(* No error *)
	IF bError=FALSE THEN
		(*Event : Alarm*)
		IF strEventType='ALARM' THEN
			(*Set Alarm*)
			IF bEventSet=TRUE THEN
				GV_Events.aEventGroup[iEventGroup].aAlarm[iIdEvent].fbAlarm.Raise(0);
			ELSE
				GV_Events.aEventGroup[iEventGroup].aAlarm[iIdEvent].fbAlarm.Confirm(0);
				GV_Events.aEventGroup[iEventGroup].aAlarm[iIdEvent].fbAlarm.Clear(0,FALSE);
			END_IF
		END_IF
		(*Event : Message*)
		IF strEventType='MESSAGE' THEN
			GV_Events.aEventGroup[iEventGroup].aMessage[iIdEvent].fbMessage.Send(0);
		END_IF
		(*Event : OpMessage*)
		IF strEventType='OpMESSAGE' THEN
			(*Set Alarm*)
			IF bEventSet=TRUE THEN
				GV_Events.aEventGroup[iEventGroup].aOpMessage[iIdEvent].fbAlarm.Raise(0);
			ELSE
				GV_Events.aEventGroup[iEventGroup].aOpMessage[iIdEvent].fbAlarm.Confirm(0);
				GV_Events.aEventGroup[iEventGroup].aOpMessage[iIdEvent].fbAlarm.Clear(0,FALSE);
			END_IF
		END_IF
	END_IF

METHOD M_Event_Group_State
VAR_INPUT
	(** INT **)
	iEventGroup : INT ;
END_VAR
VAR_OUTPUT
	(** FLAG **)
	bEventPresence : BOOL ;
END_VAR
VAR
	(** INT **)
	iLoop : INT ;
END_VAR
//-----------------------------------------------------------------------------------------
//
//                  			M_Event_Group_State
//
//							Etat du groupe d'évènements  			
//-----------------------------------------------------------------------------------------
//
//Auteur: G.GOETZ (inspired by S.MANTZER)
//Création: 23.01.2026
//Dernière modification : 23.01.2026 (G.GOETZ)
//       			
//-----------------------------------------------------------------------------------------
//
//     							Liste des modifications  	
//
// 23.01.2026 (G.GOETZ) -> Création		
//-----------------------------------------------------------------------------------------

(* Initialized variables *)
bEventPresence:=FALSE;

(*Check if alarm activated in Group xx*)
FOR iLoop:=1 TO GV_Events.iMaxAlarms BY 1 DO
	IF GV_Events.aEventGroup[iEventGroup].aAlarm[iLoop].fbAlarm.eConfirmationState=2 THEN
		bEventPresence:=TRUE;
	END_IF;
END_FOR;
END_METHOD

END_FUNCTION_BLOCK

// ---- 02_Events/03_POUs/02_FBs/FB_Init_Call_Events.TcPOU
FUNCTION_BLOCK FB_Init_Call_Events
VAR_INPUT
END_VAR
VAR_OUTPUT
END_VAR
VAR
	(** FB **)
	fbInitEvents : FB_Init_Events ;
	fbEventGroupAssignement : FB_Event_Group_Number_Assignement ;
END_VAR

//-----------------------------------------------------------------------------------------
//
//                  			FB_Init_Call_Events
//
//					Gestion initialisation appel des évènements  			
//-----------------------------------------------------------------------------------------
//
//Auteur: G.GOETZ (inspired by S.MANTZER)
//Création: 21.01.2026
//Dernière modification : 21.01.2026 (G.GOETZ)
//       			
//-----------------------------------------------------------------------------------------
//
//     							Liste des modifications  	
//
// 21.01.2026 (G.GOETZ) -> Création		
//-----------------------------------------------------------------------------------------

// Alarms and Messages init
// Call first Event because we need to call one Event in the GUID to have it into .xml file
// Event group number assignment
fbEventGroupAssignement(iEventGroup:=GV_Events.iEventGroupCallEvent);
GV_Events.aEventGroup[GV_Events.iEventGroupCallEvent].aAlarm[1].fbAlarm.CreateEx(TC_Events.EventsAlarms.Alarm1,TRUE,0);
GV_Events.aEventGroup[GV_Events.iEventGroupCallEvent].aMessage[1].fbMessage.CreateEx(TC_Events.EventsMessages.Message1,0);

fbInitEvents(iEventGroup:=GV_Events.iEventGroupCallEvent, strEventType:='ALARM', strEventGuid:='784AC907-376D-4A8E-8897-3F447F113731', tcEventSeverity:=2);
fbInitEvents(iEventGroup:=GV_Events.iEventGroupCallEvent, strEventType:='MESSAGE', strEventGuid:='8930F18E-C6C1-418F-90B9-F30993F2C9E2', tcEventSeverity:=0);

END_FUNCTION_BLOCK

// ---- 02_Events/03_POUs/02_FBs/FB_Init_Events.TcPOU
FUNCTION_BLOCK FB_Init_Events
VAR_INPUT
	(** STRING **)	
	strEventType : STRING[20] ; // Type of the Event (ALARM or MESSAGE)
	strEventGuid : STRING[36] ; // Guid of the Event
	
	(** INT **)
	iEventGroup : INT ; // Event group number

	(** TC **)
	tcEventSeverity : TcEventSeverity ;
END_VAR
VAR_OUTPUT
END_VAR
VAR
	(** UDINT **)
	uEventLoop : UDINT ; // Use in a FOR Loop
	uAlarmLength : UDINT ; // Alarm Length
	uMessageLength : UDINT ; // Message Length	
	uOpMessageLength : UDINT ; // Operator Message Length
	uIdEventStart : UDINT; // Event number start
	
	(** INT **)
	iIdStart : INT :=0 ; // Start number
	iFctState : INT ; // State of the function
	
	(** FLAG **)
	bError : BOOL ; // Error

	(** TC **)
	tcEventData : TcEventEntry ;		
END_VAR

//-----------------------------------------------------------------------------------------
//
//                  			FB_Init_Events
//
//					Gestion initialisation des évènements  			
//-----------------------------------------------------------------------------------------
//
//Auteur: G.GOETZ (inspired by S.MANTZER)
//Création: 21.01.2026
//Dernière modification : 21.01.2026 (G.GOETZ)
//       			
//-----------------------------------------------------------------------------------------
//
//     							Liste des modifications  	
//
// 21.01.2026 (G.GOETZ) -> Création		
//-----------------------------------------------------------------------------------------

(* Initialized variables *)
	bError:=FALSE;
	iIdStart:=UDINT_TO_INT(uIdEventStart);
	uAlarmLength:=INT_TO_UDINT(GV_Events.iMaxAlarms);
	uMessageLength:=INT_TO_UDINT(GV_EVENTS.iMaxMessages);
	uOpMessageLength:=INT_TO_UDINT(GV_EVENTS.iMaxOPMessages);
	uIdEventStart:=1;

(* Check EVENT GROUP, ID event, EVENT TYPE *)
	IF (iEventGroup <=0 OR iEventGroup>GV_events.iMaxEventGroup) THEN
		GV_Events.aEventGroup[GV_Events.iEventGroupCallEvent].aMessage[5].fbMessage.Send(0); // Set MESSAGE 5 (FB_EVENT EVENT GROUP number error)
		bError:=TRUE;
	ELSE
		IF  (strEventType<>'ALARM' AND strEventType<>'MESSAGE' AND strEventType<>'OpMESSAGE') THEN
			GV_Events.aEventGroup[GV_Events.iEventGroupCallEvent].aMessage[4].fbMessage.Send(0); // Set Message 4 (FB_EVENT Event type error)
			bError:=TRUE;
		ELSE
			IF ((uIdEventStart<=0 OR iIdStart>GV_Events.iMaxAlarms) AND strEventType='ALARM') THEN
				GV_Events.aEventGroup[GV_Events.iEventGroupCallEvent].aMessage[2].fbMessage.Send(0); // Set Message 2 (FB_EVENT Alarm number error)
				bError:=TRUE;
			END_IF
			IF ((uIdEventStart<=0 OR iIdStart>GV_Events.iMaxMessages) AND strEventType='MESSAGE') THEN
				GV_Events.aEventGroup[GV_Events.iEventGroupCallEvent].aMessage[3].fbMessage.Send(0); // Set Message 3 (FB_EVENT Message number error)
				bError:=TRUE;
			END_IF	
			IF ((uIdEventStart<=0 OR iIdStart>GV_Events.iMaxOPMessages) AND strEventType='OpMESSAGE') THEN
				GV_Events.aEventGroup[GV_Events.iEventGroupCallEvent].aMessage[6].fbMessage.Send(0); // Set Message 6 (FB_EVENT Operator Message number error)
				bError:=TRUE;
			END_IF
		END_IF
	END_IF

(* No error *)
	IF bError=FALSE THEN
		(*Check if Alarm  to initialize*)
		IF strEventType='ALARM' THEN
			(*Alarm init loop*)
			FOR uEventLoop:=1 TO uAlarmLength BY 1 DO
				tcEventData.uuidEventClass:=STRING_TO_GUID(strEventGuid);
				tcEventData.nEventId:=((uEventLoop+uIdEventStart)-1);
				tcEventData.eSeverity:=tcEventSeverity;
				GV_Events.aEVentGroup[iEventGroup].aAlarm[tcEventData.nEventId].fbAlarm.CreateEx(tcEventData,TRUE,0);
			END_FOR
		END_IF 
		(*Check if Message  to initialize*)
		IF strEventType='MESSAGE' THEN
			(*Alarm init loop*)
			FOR uEventLoop:=1 TO uMessageLength BY 1 DO
				tcEventData.uuidEventClass:=STRING_TO_GUID(strEventGuid);
				tcEventData.nEventId:=((uEventLoop+uIdEventStart)-1);
				tcEventData.eSeverity:=tcEventSeverity;
				GV_Events.aEVentGroup[iEventGroup].aMessage[tcEventData.nEventId].fbMessage.CreateEx(tcEventData,0);
			END_FOR
		END_IF 	
		(*Check if OpMessage  to initialize*)
		IF strEventType='OpMESSAGE' THEN
			(*Alarm init loop*)
			FOR uEventLoop:=1 TO uOpMessageLength BY 1 DO
				tcEventData.uuidEventClass:=STRING_TO_GUID(strEventGuid);
				tcEventData.nEventId:=((uEventLoop+uIdEventStart)-1);
				tcEventData.eSeverity:=tcEventSeverity;
				GV_Events.aEVentGroup[iEventGroup].aOpMessage[tcEventData.nEventId].fbAlarm.CreateEx(tcEventData,TRUE,0);
			END_FOR
		END_IF 
	END_IF

END_FUNCTION_BLOCK

// ---- 03_Operating_Mode/03_POUs/01_PRGs/PRG_OpMode.TcPOU
PROGRAM PRG_OpMode
VAR
	(** R_TRIG **)
		rtInitCycleDone : R_TRIG ;
		rtInitRequest : R_TRIG ;
END_VAR

//-----------------------------------------------------------------------------------------
//
//                  				PRG_OpMode
//
//								Programme op Mode			
//-----------------------------------------------------------------------------------------
//
//Auteur: G.GOETZ
//Création: 20.02.2026
//Dernière modification : 20.02.2026 (G.GOETZ)
//       			
//-----------------------------------------------------------------------------------------
//
//     							Liste des modifications  	
//
// 20.02.2026 (G.GOETZ) -> Création	
//-----------------------------------------------------------------------------------------

(** EVENTS **)

(** REQUEST **)
	rtInitCycleDone(CLK:=GV_Cycle.bInitCycleDone);
	rtInitRequest(CLK:=GV_Cycle.bInitRequest);
	
	(* Init *)
		IF GV_HMI.rtINIT.Q OR rtInitRequest.Q OR (GV_OpMode.eOpMode=ENUM_OpMode.AUTO AND ((NOT GV_Cycle.bCycleInProgress) OR (GV_Cycle.bCycleInProgress AND (NOT GV_Cycle.bStartStop))) AND (NOT GV_Cycle.bInitCycleDone)) THEN
			GV_OpMode.eOpModeRequest:=ENUM_OpMode.INIT;
		END_IF
	(* Auto *)
		IF (GV_HMI.rtAUTO.Q (*OR rtInitCycleDone.Q*)) AND GV_Cycle.bInitCycleDone THEN
			GV_OpMode.eOpModeRequest:=ENUM_OpMode.AUTO;
		END_IF
	(* Manu *)
		IF GV_HMI.rtMANU.Q THEN
			GV_OpMode.eOpModeRequest:=ENUM_OpMode.MANU;
		END_IF

(** AUTHORIZATION **)
		(* Init *)
			GV_OpMode.bInitAllowed:=GV_General.bSafety AND GV_General.bPower AND GV_General.bAir AND (*GV_Axes.bAxisAllOperational AND*) GV_Axes.bAxisAllNotMoving AND (((NOT GV_Cycle.bCycleInProgress) OR (GV_Cycle.bCycleInProgress AND (NOT GV_Cycle.bStartStop))) OR GV_Cycle.eCycleStep=ENUM_Cycle_Step.Error);
		(* Auto *)
			GV_OpMode.bAutoAllowed:=GV_General.bSafety AND GV_General.bPower AND GV_General.bAir AND (*GV_Axes.bAxisAllOperational AND*) GV_Axes.bAxisAllNotMoving AND GV_Cycle.bInitCycleDone;
		(* Manu *)
			GV_OpMode.bManuAllowed:=(*GV_General.bSafety AND*) GV_General.bPower AND GV_General.bAir AND (*GV_Axes.bAxisAllOperational AND*) GV_Axes.bAxisAllNotMoving AND ((NOT GV_Cycle.bCycleInProgress) OR GV_Cycle.eCycleStep=ENUM_Cycle_Step.Error);
	
(** OPMODE **)
	(*Transition*)
		IF GV_OpMode.eOpModeRequest<>GV_OpMode.eOpMode THEN 
			CASE GV_OpMode.eOpModeRequest OF
		
				ENUM_OpMode.INIT :
					IF GV_OpMode.bInitAllowed THEN
						GV_HMI.stAxes.iVelocityPourcent:=0; // Velocity 0%
						//GV_Cycle.bInitCycleDone:=FALSE;
						GV_OpMode.eOpMode:=ENUM_OpMode.INIT;
					END_IF
		
				ENUM_OpMode.AUTO :
					IF GV_OpMode.bAutoAllowed THEN
						GV_HMI.stAxes.iVelocityPourcent:=0; // Velocity 0%
						GV_OpMode.eOpMode:=ENUM_OpMode.AUTO;
					END_IF
		
				ENUM_OpMode.MANU :
					IF GV_OpMode.bManuAllowed THEN
						GV_HMI.stAxes.iVelocityPourcent:=0; // Velocity 0%
						GV_OpMode.eOpMode:=ENUM_OpMode.MANU;
					END_IF
		
			END_CASE
		END_IF
	(*InProgress*)
 		CASE GV_OpMode.eOpMode OF
  		
//  			ENUM_OpMode.INIT :
//  			 IF (NOT GV_General.bSafety) OR (NOT GV_General.bPower) OR (NOT GV_General.bAir) (*OR (NOT GV_Axes.bAxisAllOperational)*) THEN
//  				 GV_OpMode.eOpMode:=ENUM_OpMode.None;
//  			 END_IF
//  		
//  			ENUM_OpMode.AUTO :
//  			 IF ((NOT GV_General.bSafety) OR (NOT GV_General.bPower) OR (NOT GV_General.bAir) (*OR (NOT GV_Axes.bAxisAllOperational)*)) OR ((NOT GV_Cycle.bCycleInProgress) AND (NOT GV_Cycle.bInitCycleDone)) THEN
//  				 GV_OpMode.eOpMode:=ENUM_OpMode.None;
//  			 END_IF
//  			 
  			ENUM_OpMode.MANU :
  			 IF (*(NOT GV_General.bSafety) OR*) (NOT GV_General.bPower) OR (NOT GV_General.bAir) (*OR (NOT GV_Axes.bAxisAllOperational)*) THEN
  				 GV_OpMode.eOpMode:=ENUM_OpMode.None;
  			 END_IF
 			 
  		END_CASE

END_PROGRAM

// ---- 04_Lamps_Lights/03_POUs/01_PRGs/PRG_Lamps_Lights.TcPOU
PROGRAM PRG_Lamps_Lights
VAR
	(** DINT **)
	diLightsTimer : DINT ;  // Timer lights from HMI convert in DINT
	
	(** INT **)
	iDoorLoop : INT := 0 ; // INT use in a FOR Loop
	
	(** FLAG**)
	bLightsOut : BOOL := FALSE ; // Output to turn ON the lights
	
	(** FB **)
	TonLights : TON ; // Lights timer
END_VAR

//-----------------------------------------------------------------------------------------
//
//                  				PRG_Lamps_Lights
//
//							Gestion des voyants et lumières     			
//-----------------------------------------------------------------------------------------
//
//Auteur: G.GOETZ
//Création: 13.01.2026
//Dernière modification : 20.02.2026 (G.GOETZ)
//       			
//-----------------------------------------------------------------------------------------
//
//     							Liste des modifications  	
//
// 13.01.2026 (G.GOETZ) -> Création		
// 20.02.2026 (G.GOETZ) -> Ajout AUTO/MANU/INIT
//-----------------------------------------------------------------------------------------

(** LIGHTS **)
	(* Timer lights from HMI *)
		diLightsTimer:=INT_TO_DINT(GV_HMI.stLampsLights.iLightsTimer);
		IF diLightsTimer<1 THEN // Mini = 1
			diLightsTimer:=INT_TO_DINT(1);
		END_IF
	(* Light ON /OFF *)
		FOR iDoorLoop:=1 TO GV_Doors.iMaxDoors BY 1 DO
			IF GV_Doors.aId[iDoorLoop].rtButtonUnlockTrig.Q THEN //when door unlock request
				GV_HMI.stLampsLights.bLightsButton:=TRUE;
			END_IF
		END_FOR
		TonLights(IN:=(GV_HMI.stLampsLights.bLightsWithTimer AND bLightsOut),PT:=DINT_TO_TIME(diLightsTimer*60000)); // With timer and lights ON
		IF TonLights.Q THEN
			GV_HMI.stLampsLights.bLightsButton:=FALSE;
		END_IF
		IF GV_HMI.stLampsLights.bLightsButton THEN // Lights ON or OFF
			bLightsOut:=TRUE;
		ELSE
			bLightsOut:=FALSE;	
		END_IF
		GV_IO.doMagazineLight:=bLightsOut; // Lights output
		
(** LAMPS **)
	(* Init *)
		IF GV_OpMode.eOpMode=ENUM_OpMode.INIT THEN // InProgress
			GV_HMI.stLampsLights.bLampInit:=TRUE;
		ELSIF GV_OpMode.eOpModeRequest=ENUM_OpMode.INIT THEN // Request
			GV_HMI.stLampsLights.bLampInit:=GV_General.bIsBlinking05s;
		ELSE
			GV_HMI.stLampsLights.bLampInit:=FALSE;
		END_IF
	(* Auto *)
		IF GV_OpMode.eOpMode=ENUM_OpMode.AUTO THEN // InProgress
			GV_HMI.stLampsLights.bLampAuto:=TRUE;
		ELSIF GV_OpMode.eOpModeRequest=ENUM_OpMode.AUTO THEN // Request
			GV_HMI.stLampsLights.bLampAuto:=GV_General.bIsBlinking05s;
		ELSE
			GV_HMI.stLampsLights.bLampAuto:=FALSE;
		END_IF
	(* Manu *)
		IF GV_OpMode.eOpMode=ENUM_OpMode.MANU THEN // InProgress
			GV_HMI.stLampsLights.bLampManu:=TRUE;
		ELSIF GV_OpMode.eOpModeRequest=ENUM_OpMode.MANU THEN // Request
			GV_HMI.stLampsLights.bLampManu:=GV_General.bIsBlinking05s;
		ELSE
			GV_HMI.stLampsLights.bLampManu:=FALSE;
		END_IF
		
	(* Acknowledgement *)
		IF GV_HMI.bAlarm THEN
			GV_HMI.stLampsLights.bLampAck:=GV_General.bIsBlinking05s;
		ELSE
			GV_HMI.stLampsLights.bLampAck:=FALSE;
		END_IF
		
	(* Start *)
		IF GV_Cycle.bStartStop THEN // InProgress
			GV_HMI.stLampsLights.bLampStartCycle:=TRUE;
		//ELSIF GV_Cycle.bStartRequest THEN // Request
		//	GV_HMI.stLampsLights.bLampStartCycle:=GV_General.bIsBlinking05s;
		ELSE
			GV_HMI.stLampsLights.bLampStartCycle:=FALSE;
		END_IF
	(* Stop *)
		IF (NOT GV_Cycle.bStartStop) THEN // InProgress
			GV_HMI.stLampsLights.bLampStopCycle:=TRUE;
		//ELSIF GV_Cycle.bStopRequest THEN // Request
		//	GV_HMI.stLampsLights.bLampStopCycle:=GV_General.bIsBlinking05s;
		ELSE
			GV_HMI.stLampsLights.bLampStopCycle:=FALSE;
		END_IF
	
	(* Manipulator Gripper Close Manual Enable *)
		GV_HMI.stLampsLights.bLampManuManipGripperCloseEnable:=GV_Tool_Magazine.stManipulator.bAuthorizationManuGripperClose;
	(* Manipulator Gripper Open Manual Enable *)
		GV_HMI.stLampsLights.bLampManuManipGripperOpenEnable:=GV_Tool_Magazine.stManipulator.bAuthorizationManuGripperOpen;

	(* Intermediate door *)
		(*Cyltronic Rest Manual Enable*)
			GV_HMI.stLampsLights.bLampManuCyltronicRestEnable:=GV_Cyltronic.aId[1].bAuthorizationManuCyltronicRest;
		(*Cyltronic Work Manual Enable*)
			GV_HMI.stLampsLights.bLampManuCyltronicWorkEnable:=GV_Cyltronic.aId[1].bAuthorizationManuCyltronicWork;
	
	(*Axis X Operationnal*)
		GV_HMI.stLampsLights.bLampAxisXOperationnal:=GV_Axes.stAxisX.stDriveAx8206.AxisRef.Status.Operational;
	(*Axis Y Operationnal*)
		GV_HMI.stLampsLights.bLampAxisYOperationnal:=GV_Axes.stAxisY.stDriveAx8206.AxisRef.Status.Operational;
	(*Axis Z Operationnal*)
		GV_HMI.stLampsLights.bLampAxisZOperationnal:=GV_Axes.stAxisZ.stDriveAx8206.AxisRef.Status.Operational;
	(*Axis Arm Operationnal*)
		GV_HMI.stLampsLights.bLampAxisArmOperationnal:=GV_Axes.stAxisArm.stDriveAx8206.AxisRef.Status.Operational;
		
	(*Choice Axis X*)
		IF GV_Axes.eJogAxisSelect=ENUM_Axis_Select.X THEN // InProgress
			GV_HMI.stLampsLights.bLampJogAxisX:=TRUE;
		ELSIF GV_Axes.eJogAxisRequest=ENUM_Axis_Select.X THEN // Request
			GV_HMI.stLampsLights.bLampJogAxisX:=GV_General.bIsBlinking05s;
		ELSE
			GV_HMI.stLampsLights.bLampJogAxisX:=FALSE;
		END_IF
	(*Choice Axis Z*)
		IF GV_Axes.eJogAxisSelect=ENUM_Axis_Select.Z THEN // InProgress
			GV_HMI.stLampsLights.bLampJogAxisZ:=TRUE;
		ELSIF GV_Axes.eJogAxisRequest=ENUM_Axis_Select.Z THEN // Request
			GV_HMI.stLampsLights.bLampJogAxisZ:=GV_General.bIsBlinking05s;
		ELSE
			GV_HMI.stLampsLights.bLampJogAxisZ:=FALSE;
		END_IF
	(*Choice Axis Y*)
		IF GV_Axes.eJogAxisSelect=ENUM_Axis_Select.Y THEN // InProgress
			GV_HMI.stLampsLights.bLampJogAxisY:=TRUE;
		ELSIF GV_Axes.eJogAxisRequest=ENUM_Axis_Select.Y THEN // Request
			GV_HMI.stLampsLights.bLampJogAxisY:=GV_General.bIsBlinking05s;
		ELSE
			GV_HMI.stLampsLights.bLampJogAxisY:=FALSE;
		END_IF
	(*Choice Axis Arm*)
		IF GV_Axes.eJogAxisSelect=ENUM_Axis_Select.Arm THEN // InProgress
			GV_HMI.stLampsLights.bLampJogAxisArm:=TRUE;
		ELSIF GV_Axes.eJogAxisRequest=ENUM_Axis_Select.Arm THEN // Request
			GV_HMI.stLampsLights.bLampJogAxisArm:=GV_General.bIsBlinking05s;
		ELSE
			GV_HMI.stLampsLights.bLampJogAxisArm:=FALSE;
		END_IF
		
	(*Referencing Axis None*)
		IF GV_Axes.eRefAxisSelect=ENUM_Axis_Select.None THEN // InProgress
			GV_HMI.stLampsLights.bLampEnMinSoftPosLimit:=FALSE;
			GV_HMI.stLampsLights.bLampEnMaxSoftPosLimit:=FALSE;
		END_IF
	(*Referencing Axis X*)
		IF GV_Axes.eRefAxisSelect=ENUM_Axis_Select.X THEN // InProgress
			GV_HMI.stLampsLights.bLampRefAxisX:=TRUE;
			IF GV_Axes.stAxisX.bReadEnMinSoftPosLimit THEN // Min Soft Limit Enable
				GV_HMI.stLampsLights.bLampEnMinSoftPosLimit:=TRUE;
			ELSE
				GV_HMI.stLampsLights.bLampEnMinSoftPosLimit:=FALSE;
			END_IF
			IF GV_Axes.stAxisX.bReadEnMaxSoftPosLimit THEN // Max Soft Limit Enable
				GV_HMI.stLampsLights.bLampEnMaxSoftPosLimit:=TRUE;
			ELSE
				GV_HMI.stLampsLights.bLampEnMaxSoftPosLimit:=FALSE;
			END_IF
		ELSIF GV_Axes.eRefAxisRequest=ENUM_Axis_Select.X THEN // Request
			GV_HMI.stLampsLights.bLampRefAxisX:=GV_General.bIsBlinking05s;
		ELSE
			GV_HMI.stLampsLights.bLampRefAxisX:=FALSE;
		END_IF
	(*Referencing Axis Y*)
		IF GV_Axes.eRefAxisSelect=ENUM_Axis_Select.Y THEN // InProgress
			GV_HMI.stLampsLights.bLampRefAxisY:=TRUE;
			IF GV_Axes.stAxisY.bReadEnMinSoftPosLimit THEN // Min Soft Limit Enable
				GV_HMI.stLampsLights.bLampEnMinSoftPosLimit:=TRUE;
			ELSE
				GV_HMI.stLampsLights.bLampEnMinSoftPosLimit:=FALSE;
			END_IF
			IF GV_Axes.stAxisY.bReadEnMaxSoftPosLimit THEN // Max Soft Limit Enable
				GV_HMI.stLampsLights.bLampEnMaxSoftPosLimit:=TRUE;
			ELSE
				GV_HMI.stLampsLights.bLampEnMaxSoftPosLimit:=FALSE;
			END_IF
		ELSIF GV_Axes.eRefAxisRequest=ENUM_Axis_Select.Y THEN // Request
			GV_HMI.stLampsLights.bLampRefAxisY:=GV_General.bIsBlinking05s;
		ELSE
			GV_HMI.stLampsLights.bLampRefAxisY:=FALSE;
		END_IF
	(*Referencing Axis Z*)
		IF GV_Axes.eRefAxisSelect=ENUM_Axis_Select.Z THEN // InProgress
			GV_HMI.stLampsLights.bLampRefAxisZ:=TRUE;
			IF GV_Axes.stAxisZ.bReadEnMinSoftPosLimit THEN // Min Soft Limit Enable
				GV_HMI.stLampsLights.bLampEnMinSoftPosLimit:=TRUE;
			ELSE
				GV_HMI.stLampsLights.bLampEnMinSoftPosLimit:=FALSE;
			END_IF
			IF GV_Axes.stAxisZ.bReadEnMaxSoftPosLimit THEN // Max Soft Limit Enable
				GV_HMI.stLampsLights.bLampEnMaxSoftPosLimit:=TRUE;
			ELSE
				GV_HMI.stLampsLights.bLampEnMaxSoftPosLimit:=FALSE;
			END_IF
		ELSIF GV_Axes.eRefAxisRequest=ENUM_Axis_Select.Z THEN // Request
			GV_HMI.stLampsLights.bLampRefAxisZ:=GV_General.bIsBlinking05s;
		ELSE
			GV_HMI.stLampsLights.bLampRefAxisZ:=FALSE;
		END_IF
	(*Referencing Axis Arm*)
		IF GV_Axes.eRefAxisSelect=ENUM_Axis_Select.Arm THEN // InProgress
			GV_HMI.stLampsLights.bLampRefAxisArm:=TRUE;
			IF GV_Axes.stAxisArm.bReadEnMinSoftPosLimit THEN // Min Soft Limit Enable
				GV_HMI.stLampsLights.bLampEnMinSoftPosLimit:=TRUE;
			ELSE
				GV_HMI.stLampsLights.bLampEnMinSoftPosLimit:=FALSE;
			END_IF
			IF GV_Axes.stAxisArm.bReadEnMaxSoftPosLimit THEN // Max Soft Limit Enable
				GV_HMI.stLampsLights.bLampEnMaxSoftPosLimit:=TRUE;
			ELSE
				GV_HMI.stLampsLights.bLampEnMaxSoftPosLimit:=FALSE;
			END_IF
		ELSIF GV_Axes.eRefAxisRequest=ENUM_Axis_Select.Arm THEN // Request
			GV_HMI.stLampsLights.bLampRefAxisArm:=GV_General.bIsBlinking05s;
		ELSE
			GV_HMI.stLampsLights.bLampRefAxisArm:=FALSE;
		END_IF
		
	(*Project Backup Enable*)
		GV_HMI.stLampsLights.bLampBackupProjectEnable:=GV_General.bBackupProjectAuthorization;
	(*Init Data Enable*)
		GV_HMI.stLampsLights.bLampDataInitEnable:=GV_General.bInitDataAuthorization;			
	(*Export Data Enable*)
		GV_HMI.stLampsLights.bLampDataExportEnable:=GV_General.bExportDataAuthorization;	
	(*Import Data Enable*)
		GV_HMI.stLampsLights.bLampDataImportEnable:=GV_General.bImportDataAuthorization;	
	(*Export Alarms Enable*)
		GV_HMI.stLampsLights.bLampAlarmsExportEnable:=GV_General.bExportAlarmsAuthorization;	
	(*Export Messages Enable*)
		GV_HMI.stLampsLights.bLampMessagesExportEnable:=GV_General.bExportMessagesAuthorization;
	(* Save Settings Enable *)
		GV_HMI.stLampsLights.bLampSettingsSaveEnable:=GV_General.bSettingSaveAuthorization;
		
	(*Teach Location Enable*)
		GV_HMI.stLampsLights.bLampTeachLocationEnable:=GV_Tool_Magazine.bAuthorizationTeachLocation;
	(*Teach Line Enable*)
		GV_HMI.stLampsLights.bLampTeachRackEnable:=GV_Tool_Magazine.bAuthorizationTeachRack;
	(*Teach AllTop Enable*)
		GV_HMI.stLampsLights.bLampTeachAllTopEnable:=GV_Tool_Magazine.bAuthorizationTeachAllTop;
	(*Teach AllBottom Enable*)
		GV_HMI.stLampsLights.bLampTeachAllBottomEnable:=GV_Tool_Magazine.bAuthorizationTeachAllBottom;
	(*Teach Positions Enable *)
		GV_HMI.stLampsLights.bLampTeachPositionsEnable:=GV_Tool_Magazine.bAuthorizationTeachPositions;
		
	(*Reboot Enable*)
		GV_HMI.stLampsLights.bLampRebootEnable:=GV_General.bRebootAuthorization;
	(*Shutdown Enable*)
		GV_HMI.stLampsLights.bLampShutdownEnable:=GV_General.bShutdownAuthorization;

END_PROGRAM

// ---- 05_Fans/03_POUs/01_PRGs/PRG_Fans.TcPOU
PROGRAM PRG_Fans
VAR
	(** REAL **)
		rProportionnal: REAL := 0 ;	// kP for the Fan regulation

	(** WORD **)
		wPT100ArmorValue : WORD ;
		wPT100ArmorValue1 : WORD ;
		wPT100ArmorValue2 : WORD ;

	(** INT **)
		iFanLoop : INT := 0 ; // INT use in a FOR Loop
	
	(** BYTE **)
		bPT100ArmorValue1 : BYTE ;
		bPT100ArmorValue2 : BYTE ;
	
	(** FB **)
		FbFan : FB_Fan ;
		fbEventGroupAssignement : FB_Event_Group_Number_Assignement ;
END_VAR

//-----------------------------------------------------------------------------------------
//
//                  				PRG_Fans
//
//			Paramétrage ventilateur(s) + Appel Gestion ventilateur(s)  			
//-----------------------------------------------------------------------------------------
//
//Auteur: G.GOETZ
//Création: 20.01.2026
//Dernière modification : 20.01.2026 (G.GOETZ)
//       			
//-----------------------------------------------------------------------------------------
//
//     							Liste des modifications  	
//
// 20.01.2026 (G.GOETZ) -> Création		
//-----------------------------------------------------------------------------------------

(** MAGAZINE ARMOR FAN **)
	GV_Fans.aId[1].bPresence:=TRUE; // Fan presence or not
	fbEventGroupAssignement(iEventGroup:=GV_Fans.aId[1].iEventGroup);
	GV_Fans.aId[1].iIdHMI:=1; // Number for events on HMI
	GV_Fans.aId[1].eFanType:=ENUM_Fan_Type.PWM; // Fan type
	GV_Fans.aId[1].uPwmPeriod:=40; // PWM period 100ns = 10kHz
	GV_Fans.aId[1].uMinSpeed:=1000; // Min speed 1000tr/min
	GV_Fans.aId[1].uMaxSpeed:=8500; // Max speed 8500tr/min
	GV_Fans.aId[1].uMinPwm:=10; // Min Pwm = 10% at min speed
	GV_Fans.aId[1].uMaxPwm:=100; // Max Pwm = 95% at max speed
	GV_Fans.aId[1].rTempStart:=30.0; // Temp in °C to start the fan
	GV_Fans.aId[1].rTempMax:=45.0; // Temp in °C for max speed of the fan
	GV_IO.pwmMagazineArmorFanOutput:=LREAL_TO_UINT(UINT_TO_LREAL(GV_Fans.aId[1].uPwmOutput)*200); // PWM output (0-65535) -> (0-20000)
	GV_IO.pwmMagazineArmorFanPeriod:=GV_Fans.aId[1].uPwmPeriod; // PWM perod
	(* Speed Set *)
		(* PT100 Armor *)
			wPT100ArmorValue1:=GV_CNC.stFanucData.stCncMagazine.wiPT100ArmorValue; // Temp from CNC
			//MSB  
			bPT100ArmorValue1:=WORD_TO_BYTE(SHR(wPT100ArmorValue1,8));
			//LSB
			bPT100ArmorValue2:=WORD_TO_BYTE(wPT100ArmorValue1 AND 16#FF);
			wPT100ArmorValue:=(SHL(BYTE_TO_WORD(bPT100ArmorValue2),8) OR BYTE_TO_WORD(bPT100ArmorValue1));
		GV_Fans.rTempArmor:=WORD_TO_REAL(wPT100ArmorValue/10); // Temp convert from CNC
		IF GV_Fans.rTempArmor<=-1 OR GV_Fans.rTempArmor>=1 THEN
			GV_Fans.rTempArmorFiltered:=GV_Fans.rTempArmorFiltered+0.05*(GV_Fans.rTempArmor-GV_Fans.rTempArmorFiltered); // Temp Filtered
		ELSE
			GV_Fans.rTempArmorFiltered:=0;
		END_IF
		IF GV_Fans.rTempArmorFiltered<=GV_Fans.aId[1].rTempStart THEN
			GV_Fans.aId[1].uSpeedSet:=GV_Fans.aId[1].uMinSpeed; // Speed command (Min speed)
		ELSIF GV_Fans.rTempArmorFiltered>=GV_Fans.aId[1].rTempMax THEN
			GV_Fans.aId[1].uSpeedSet:=GV_Fans.aId[1].uMaxSpeed; // Speed command (Max speed)
		ELSE
		   IF GV_Fans.aId[1].rTempMax>GV_Fans.aId[1].rTempStart THEN
				rProportionnal:=(GV_Fans.rTempArmorFiltered-GV_Fans.aId[1].rTempStart)/(GV_Fans.aId[1].rTempMax-GV_Fans.aId[1].rTempStart);
				GV_Fans.aId[1].uSpeedSet:=GV_Fans.aId[1].uMinSpeed+REAL_TO_UINT(rProportionnal*(GV_Fans.aId[1].uMaxSpeed-GV_Fans.aId[1].uMinSpeed));
			ELSE
					 GV_Fans.aId[1].uSpeedSet:=GV_Fans.aId[1].uMaxSpeed;
			END_IF
		END_IF

	(*Limit*)
		IF GV_Fans.aId[1].uSpeedSet<GV_Fans.aId[1].uMinSpeed THEN
			GV_Fans.aId[1].uSpeedSet:=GV_Fans.aId[1].uMinSpeed;
		END_IF
		IF GV_Fans.aId[1].uSpeedSet>GV_Fans.aId[1].uMaxSpeed THEN
			GV_Fans.aId[1].uSpeedSet:=GV_Fans.aId[1].uMaxSpeed;
		END_IF
	
	(*Start*)
		GV_Fans.aId[1].rtStart(CLK:=GV_General.bSafety);
 		 IF GV_Fans.aId[1].rtStart.Q THEN
 			 GV_Fans.aId[1].bStart:=TRUE;
 		 END_IF
		
(** OTHER FAN **)
	//...

(** FB_Fan **)
	FOR iFanLoop:=1 TO GV_Fans.iMaxFans BY 1 DO
		FbFan(iFanNumber:=iFanLoop,StFan:=GV_Fans.aId[iFanLoop]); // Fan function block
	END_FOR

END_PROGRAM

// ---- 05_Fans/03_POUs/02_FBs/FB_Fan.TcPOU
FUNCTION_BLOCK FB_Fan
VAR_INPUT
	(** INT **)
	iFanNumber : INT ; // Number of the fan
END_VAR
VAR_OUTPUT
END_VAR
VAR_IN_OUT
	(** ST **)
	stFan : ST_Fan ;
END_VAR
VAR
	(** FB **)
	fbInitEvents : FB_Init_Events ;
	fbEventHMI : FB_Event_HMI ;
	
	tonStartMin : TON ;
	tonStartMax : TON ;
END_VAR

//-----------------------------------------------------------------------------------------
//
//                  				FB_Fan
//
//							Gestion ventilateur(s)   			
//-----------------------------------------------------------------------------------------
//
//Auteur: G.GOETZ
//Création: 20.01.2026
//Dernière modification : 27.01.2026 (G.GOETZ)
//       			
//-----------------------------------------------------------------------------------------
//
//     							Liste des modifications  	
//
// 20.01.2026 (G.GOETZ) -> Création	
// 27.01.2026 (G.GOETZ) -> Ajout gestion des alarmes/messages
//-----------------------------------------------------------------------------------------

IF stFan.bPresence THEN
		
	(** EVENTS **)
		IF GV_General.bFirstCycleTask OR GV_General.bFirstCycleSimu THEN
			(*Call first Event because we need to call one Event in the GUID to have it into .xml file*)
			GV_Events.aEventGroup[GV_Fans.aId[iFanNumber].iEventGroup].aAlarm[1].fbAlarm.CreateEx(TC_Events.FanAlarms.Alarm1,TRUE,0);
			GV_Events.aEventGroup[GV_Fans.aId[iFanNumber].iEventGroup].aOpMessage[1].fbAlarm.CreateEx(TC_Events.FanOpMessages.Message1,TRUE,0);	
			fbInitEvents(iEventGroup:=GV_Fans.aId[iFanNumber].iEventGroup,strEventType:='ALARM',strEventGuid:='77BDDCBB-B8DC-46C2-9AE2-0C0996835A2C',tcEventSeverity:=2);
			fbInitEvents(iEventGroup:=GV_Fans.aId[iFanNumber].iEventGroup,strEventType:='OpMESSAGE',strEventGuid:='7465A544-4166-4343-9B32-33A0414E8A0C',tcEventSeverity:=1);
		END_IF

	(** FAN TYPES MANAGEMENT **)

	(* 1 With PWM type *) // WIth rampe
		IF stFan.eFanType=ENUM_Fan_Type.PWM THEN

			tonStartMin(PT:=T#3S);
			tonStartMax(PT:=T#3S);
			
			(* Start Sequence *)
			IF stFan.bStart AND GV_General.bSafety THEN
				
				tonStartMin(PT:=T#3S);
				tonStartMax(PT:=T#3S);
				
				(*At Min*)
				IF (NOT tonStartMin.Q) THEN
					stFan.uPwmOutput:=0; // PWM output
				END_IF
				IF stFan.uPwmOutput=0 THEN
					tonStartMin.IN:=TRUE;
				END_IF
				
				(*At Max*)		
				IF tonStartMin.Q THEN
					stFan.uPwmOutput:=327; // PWM output 327*200=(0-65535)
				END_IF
				IF stFan.uPwmOutput=327 THEN
					tonStartMax.IN:=TRUE;
				END_IF
				
				(*Done*)
				IF tonStartMax.Q THEN
					tonStartMin.IN:=FALSE;
					tonStartMax.IN:=FALSE;
					stFan.bStart:=FALSE;
				END_IF
				
			ELSE
				stFan.bStart:=FALSE;

				tonStartMin.IN:=FALSE;
				tonStartMax.IN:=FALSE;
				
				(* Target *)
				(*Min*)
				IF stFan.uSpeedSet<=stFan.uMinSpeed THEN
					stFan.uPwmTarget:=stFan.uMinPwm; // Min% PWM
				END_IF
				(*Max*)
				IF stFan.uSpeedSet>=stFan.uMaxSpeed THEN
					stFan.uPwmTarget:=stFan.uMaxPwm; // Max% PWM
				END_IF
				(*PWM = PWMmin + (Speed - MinSpeed) × (PWMmax - PWMmin) / (Speedmax - Speedmin)*)
				IF stFan.uSpeedSet>stFan.uMinSpeed AND stFan.uSpeedSet<stFan.uMaxSpeed THEN
					stFan.uPwmTarget:=(stFan.uMinPwm+((stFan.uSpeedSet-stFan.uMinSpeed)*(stFan.uMaxPwm-stFan.uMinPwm))/(stFan.uMaxSpeed-stFan.uMinSpeed)); // X% PWM at the speed command
					stFan.uPwmTarget:=REAL_TO_UINT(stFan.uPwmTarget+0.5);
				END_IF
				IF (NOT GV_General.bSafety) THEN
					stFan.uPwmTarget:=0; // 0% PWM
				END_IF
				
				(* Command with ramp *)
				(*Accel ramp*)
				IF stFan.uPwmOutput<stFan.uPwmTarget THEN
					stFan.uPwmOutput:=MIN(stFan.uPwmOutput+GV_Fans.uRampStep1,stFan.uPwmTarget);
				END_IF
				(*Decel ramp*)
				IF stFan.uPwmOutput>stFan.uPwmTarget THEN
					stFan.uPwmOutput:=MAX(stFan.uPwmOutput-GV_Fans.uRampStep1,stFan.uPwmTarget);
				END_IF		
		
				(*Message 1 = Fan stopped*)
				IF stFan.uPwmOutput=0 THEN // Fan setpoint at 0
					GV_Events.aEventGroup[GV_Fans.aId[iFanNumber].iEventGroup].aOpMessage[1].fbAlarm.ipArguments.Clear().AddDInt(stFan.iIdHMI);
					fbEventHMI(iEventGroup:=GV_Fans.aId[iFanNumber].iEventGroup,iIdEvent:=1,strEventType:='OpMESSAGE',bEventSet:=TRUE);
				ELSE
					fbEventHMI(iEventGroup:=GV_Fans.aId[iFanNumber].iEventGroup,iIdEvent:=1,strEventType:='OpMESSAGE',bEventSet:=FALSE);			
				END_IF
			END_IF
			
		END_IF
	
//ELSE
END_IF

END_FUNCTION_BLOCK

// ---- 06_Doors/03_POUs/01_PRGs/PRG_Doors.TcPOU
PROGRAM PRG_Doors
VAR
	(** INT **)
	iDoorLoop : INT := 0 ; // INT use in a FOR Loop
	iDoorCloseLockNumber : INT := 0 ; // How many doors are close and lock
	
	(** FB **)
	fbDoor : FB_Door ;
	fbEventGroupAssignement : FB_Event_Group_Number_Assignement ;
	
	tonCycleNotProgess : TON ;
END_VAR

//-----------------------------------------------------------------------------------------
//
//                  				PRG_Doors
//
//					Paramétrage porte(s) + Appel Gestion porte(s)  			
//-----------------------------------------------------------------------------------------
//
//Auteur: G.GOETZ (inspired by S.MANTZER)
//Création: 13.01.2026
//Dernière modification : 13.01.2026 (G.GOETZ)
//       			
//-----------------------------------------------------------------------------------------
//
//     							Liste des modifications  	
//
// 13.01.2026 (G.GOETZ) -> Création		
//-----------------------------------------------------------------------------------------

(** TOOL MAGAZINE DOOR **)
	GV_Doors.aId[1].bPresence:=TRUE; // Door prensence or not
	fbEventGroupAssignement(iEventGroup:=GV_Doors.aId[1].iEventGroup);
	GV_Doors.aId[1].iIdHMI:=1; // Number for events on HMI
	GV_Doors.aId[1].eType:=ENUM_Door_Type.AutoLockButtonUnlockOn; // Door type
	GV_Doors.aId[1].bUnlockAuthorization:=GV_IO.diSafetyRelayIntermediateDoor AND ((GV_HMI.stDoors.bDoorUnlockForce OR tonCycleNotProgess.Q OR (NOT GV_Cycle.bStartStop))); // Authorization for unlock the door
	GV_Doors.aId[1].bButtonUnlock:=GV_IO.diButtonUnlockMagazineDoor; // Button for unlock the door
	GV_Doors.aId[1].bDoorOpen:=GV_IO.diMagazineDoorOpen; // Door is open
	GV_Doors.aId[1].bDoorSafetyRelay:=GV_IO.diSafetyRelayMagazineDoor; // Safety realy of the door
	GV_IO.doButtonUnlockMagazineDoorLamp:=GV_Doors.aId[1].bButtonUnlockLamp; // Lamp of the unlock button
	GV_IO.doUnlockMagazineDoor:=GV_Doors.aId[1].bUnlockOut; // Unlock the door

	tonCycleNotProgess(IN:=(NOT GV_Cycle.bCycleInProgress),PT:=T#2S);

(** OTHER DOOR **)
//...

(** FB_Door **)
	FOR iDoorLoop:=1 TO GV_Doors.iMaxDoors BY 1 DO
		fbDoor(iDoorNumber:=iDoorLoop,StDoor:=GV_Doors.aId[iDoorLoop]); // Door function block
	END_FOR

(** DOORS OK **)
	iDoorCloseLockNumber:=0; // Init the number of doors closed and locked
	FOR iDoorLoop:=1 TO GV_Doors.iMaxDoors BY 1 DO
		IF GV_Doors.aId[iDoorLoop].bDoorCloseLock THEN // How many doors are closed and locked
			iDoorCloseLockNumber:=iDoorCloseLockNumber+1;
		END_IF
	END_FOR
	
	IF iDoorCloseLockNumber=GV_Doors.iMaxDoors THEN // All doors are closed and locked
		GV_Doors.bDoorsCloseLock:=TRUE;
	ELSE
		GV_Doors.bDoorsCloseLock:=FALSE;
	END_IF
	
(** CHECK MAGAZINE REQUEST **)
// 	IF (NOT GV_Doors.bDoorsCloseLock) OR GV_Tool_Magazine.bFirstCycleCheckMagazine THEN
// 		IF GV_HMI.stMagazineCheck.iCheckCycleType=1 THEN // One Location
// 			GV_Tool_Magazine.bCheckFullMagazineRequest:=FALSE;
// 			GV_Tool_Magazine.bCheckOneMagazineRequest:=TRUE;
// 			IF GV_Tool_Magazine.stManipulator.bToolPresenceMemory THEN // Manipulator memory
// 				GV_Tool_Magazine.bCheckManipulatorMemoryRequest:=TRUE;
// 			ELSE
// 				GV_Tool_Magazine.bCheckManipulatorMemoryRequest:=FALSE;
// 			END_IF
// 			IF GV_Tool_Magazine.stArm.aGripper[1].bToolPresenceMemory THEN // Arm gripper 1 memory
// 				GV_Tool_Magazine.bCheckArmGripper1MemoryRequest:=TRUE;
// 			ELSE
// 				GV_Tool_Magazine.bCheckArmGripper1MemoryRequest:=FALSE;
// 			END_IF
// 			IF GV_Tool_Magazine.stArm.aGripper[2].bToolPresenceMemory THEN // Arm gripper 2 memory
// 				GV_Tool_Magazine.bCheckArmGripper2MemoryRequest:=TRUE;
// 			ELSE
// 				GV_Tool_Magazine.bCheckArmGripper2MemoryRequest:=FALSE;
// 			END_IF
// 			IF GV_CNC.stSpindle.bToolPresenceMemory THEN // Spindle memory
// 				GV_Tool_Magazine.bCheckSpindleMemoryRequest:=TRUE;
// 			ELSE
// 				GV_Tool_Magazine.bCheckSpindleMemoryRequest:=FALSE;
// 			END_IF
// 		ELSIF GV_HMI.stMagazineCheck.iCheckCycleType=2 THEN // Full Location
// 			GV_Tool_Magazine.bCheckFullMagazineRequest:=TRUE;
// 			GV_Tool_Magazine.bCheckOneMagazineRequest:=FALSE;
// 			GV_Tool_Magazine.bCheckManipulatorMemoryRequest:=FALSE;
// 			GV_Tool_Magazine.bCheckArmGripper1MemoryRequest:=FALSE;
// 			GV_Tool_Magazine.bCheckArmGripper2MemoryRequest:=FALSE;
// 			GV_Tool_Magazine.bCheckSpindleMemoryRequest:=FALSE;
// 		ELSE
// 			GV_Tool_Magazine.bCheckFullMagazineRequest:=FALSE;
// 			GV_Tool_Magazine.bCheckOneMagazineRequest:=FALSE;
// 			GV_Tool_Magazine.bCheckManipulatorMemoryRequest:=FALSE;
// 			GV_Tool_Magazine.bCheckArmGripper1MemoryRequest:=FALSE;
// 			GV_Tool_Magazine.bCheckArmGripper2MemoryRequest:=FALSE;
// 			GV_Tool_Magazine.bCheckSpindleMemoryRequest:=FALSE;
// 		END_IF
// 		GV_Tool_Magazine.bFirstCycleCheckMagazine:=FALSE;
// 	END_IF

GV_Tool_Magazine.bFirstCycleCheckMagazine:=FALSE;

GV_Tool_Magazine.bCheckFullMagazineRequest:=FALSE;
GV_Tool_Magazine.bCheckOneMagazineRequest:=FALSE;
			
GV_Tool_Magazine.bCheckManipulatorMemoryRequest:=FALSE;
GV_Tool_Magazine.bCheckArmGripper1MemoryRequest:=FALSE;
GV_Tool_Magazine.bCheckArmGripper2MemoryRequest:=FALSE;
GV_Tool_Magazine.bCheckSpindleMemoryRequest:=FALSE;

END_PROGRAM

// ---- 06_Doors/03_POUs/02_FBs/FB_Door.TcPOU
FUNCTION_BLOCK FB_Door
VAR_INPUT
	(** INT **)
		iDoorNumber : INT ; // Number of the door
END_VAR
VAR_OUTPUT
END_VAR
VAR_IN_OUT
	(** ST **)
		stDoor : ST_Door ;
END_VAR
VAR
	(** FB **)
		fbInitEvents : FB_Init_Events ;
		fbEventHMI : FB_Event_HMI ;
END_VAR

//-----------------------------------------------------------------------------------------
//
//                  				FB_Door
//
//								Gestion porte(s)   			
//-----------------------------------------------------------------------------------------
//
//Auteur: G.GOETZ (inspired by S.MANTZER)
//Création: 13.01.2026
//Dernière modification : 28.01.2026 (G.GOETZ)
//       			
//-----------------------------------------------------------------------------------------
//
//     							Liste des modifications  	
//
// 13.01.2026 (G.GOETZ) -> Création	
// 28.01.2026 (G.GOETZ) -> Ajout gestion voyant bouton
//-----------------------------------------------------------------------------------------

IF stDoor.bPresence THEN
		
	(** EVENTS **)
		IF GV_General.bFirstCycleTask OR GV_General.bFirstCycleSimu THEN
			(*Call first Event because we need to call one Event in the GUID to have it into .xml file*)
			GV_Events.aEventGroup[GV_Doors.aId[iDoorNumber].iEventGroup].aAlarm[1].fbAlarm.CreateEx(TC_Events.DoorAlarms.Alarm1,TRUE,0);
			GV_Events.aEventGroup[GV_Doors.aId[iDoorNumber].iEventGroup].aOpMessage[1].fbAlarm.CreateEx(TC_Events.DoorOpMessages.Message1,TRUE,0);	
			fbInitEvents(iEventGroup:=GV_Doors.aId[iDoorNumber].iEventGroup,strEventType:='ALARM',strEventGuid:='34B37164-85A5-4BB2-918B-4ED16EAF1356',tcEventSeverity:=2);
			fbInitEvents(iEventGroup:=GV_Doors.aId[iDoorNumber].iEventGroup,strEventType:='OpMESSAGE',strEventGuid:='DBCE0E6A-9DBC-4431-B292-1C122D38EFE6',tcEventSeverity:=1);
		END_IF

	(** DOOR TYPES MANAGEMENT **)
	
	(* 1 With Auto lock AND unlock button (Output OFF unlock) *)
		IF stDoor.eType=ENUM_Door_Type.AutoLockButtonUnlockOff THEN
			
			(*Unlock request*)
			stDoor.rtButtonUnlockTrig(CLK:=stDoor.bButtonUnlock); //Trigger of the button
			IF stDoor.rtButtonUnlockTrig.Q AND (NOT stDoor.bUnlockRequest) AND (NOT stDoor.bUnlockOut) THEN
				stDoor.bUnlockRequest:=TRUE;
			END_IF
			(*Unlock request acknowledgenent*)
			IF (NOT stDoor.bUnlockAuthorization) THEN // No Authorization = reset request
				stDoor.bUnlockRequestAck:=TRUE;
			END_IF
			IF stDoor.bUnlockRequestAck THEN
				stDoor.bUnlockRequest:=FALSE;
				stDoor.bUnlockRequestAck:=FALSE;
			END_IF
			
			(*Unlock door*)
			IF stDoor.bUnlockRequest AND stDoor.bUnlockAuthorization THEN
				stDoor.bUnlockOut:=FALSE;
			END_IF
			IF (NOT stDoor.bUnlockRequest) THEN
				stDoor.bUnlockOut:=TRUE;
			END_IF
			
			(*Door open*)
			IF stDoor.bDoorOpen THEN
				stDoor.bUnlockRequest:=FALSE;
			END_IF
			
			(*Door button lamp*)
			
			(*Door close and lock*)
			IF (NOT stDoor.bDoorOpen) AND stDoor.bDoorSafetyRelay AND (NOT stDoor.bUnlockOut) THEN
				stDoor.bDoorCloseLock:=TRUE;
			ELSE
				stDoor.bDoorCloseLock:=FALSE;			
			END_IF
			
			(*Message 1 = Door open*)
			IF (NOT stDoor.bDoorCloseLock) THEN // Door open
				GV_Events.aEventGroup[GV_Doors.aId[iDoorNumber].iEventGroup].aOpMessage[1].fbAlarm.ipArguments.Clear().AddDInt(stDoor.iIdHMI);
				fbEventHMI(iEventGroup:=GV_Doors.aId[iDoorNumber].iEventGroup,iIdEvent:=1,strEventType:='OpMESSAGE',bEventSet:=TRUE);
			ELSE
				fbEventHMI(iEventGroup:=GV_Doors.aId[iDoorNumber].iEventGroup,iIdEvent:=1,strEventType:='OpMESSAGE',bEventSet:=FALSE);			
			END_IF
			
		END_IF
	
	(* 2 With Auto lock AND unlock button (Output ON unlock) *)	
		IF stDoor.eType=ENUM_Door_Type.AutoLockButtonUnlockOn THEN
			
			(*Unlock request*)
			stDoor.rtButtonUnlockTrig(CLK:=stDoor.bButtonUnlock); //Trigger of the button
			IF stDoor.rtButtonUnlockTrig.Q AND (NOT stDoor.bUnlockRequest) AND (NOT stDoor.bUnlockOut) THEN
				stDoor.bUnlockRequest:=TRUE;
			END_IF
			(*Unlock request acknowledgenent*)
			IF (NOT stDoor.bUnlockAuthorization) THEN // No Authorization = reset request
				stDoor.bUnlockRequestAck:=TRUE;
			END_IF
			IF stDoor.bUnlockRequestAck THEN
				stDoor.bUnlockRequest:=FALSE;
				stDoor.bUnlockRequestAck:=FALSE;
			END_IF
			
			(*Unlock door*)
			IF stDoor.bUnlockRequest AND stDoor.bUnlockAuthorization THEN
				stDoor.bUnlockOut:=TRUE;
			END_IF
			IF (NOT stDoor.bUnlockRequest) THEN
				stDoor.bUnlockOut:=FALSE;
			END_IF
			
			(*Door open*)
			IF stDoor.bDoorOpen THEN
				stDoor.bUnlockRequest:=FALSE;
			END_IF
			
			(*Door button lamp*)
			IF stDoor.bUnlockAuthorization AND stDoor.bDoorCloseLock THEN
				stDoor.bButtonUnlockLamp:=TRUE;
			ELSE
				IF (NOT stDoor.bDoorCloseLock) THEN
					IF GV_General.bIsBlinking1s THEN
						stDoor.bButtonUnlockLamp:=TRUE;
					ELSE
						stDoor.bButtonUnlockLamp:=FALSE;				
					END_IF	
				END_IF
				IF stDoor.bUnlockRequest AND (NOT stDoor.bUnlockAuthorization) AND stDoor.bDoorCloseLock THEN
					IF GV_General.bIsBlinking05s THEN
						stDoor.bButtonUnlockLamp:=TRUE;
					ELSE
						stDoor.bButtonUnlockLamp:=FALSE;				
					END_IF	
				END_IF
				IF (NOT stDoor.bUnlockRequest) AND (NOT stDoor.bUnlockAuthorization) AND stDoor.bDoorCloseLock THEN
					stDoor.bButtonUnlockLamp:=FALSE;	
				END_IF
			END_IF
			
			(*Door close and lock*)
			IF (NOT stDoor.bDoorOpen) AND stDoor.bDoorSafetyRelay AND (NOT stDoor.bUnlockOut) THEN
				stDoor.bDoorCloseLock:=TRUE;
			ELSE
				stDoor.bDoorCloseLock:=FALSE;			
			END_IF
			
			(*Message 1 = Door open*)
			IF (NOT stDoor.bDoorCloseLock) THEN // Door open
				GV_Events.aEventGroup[GV_Doors.aId[iDoorNumber].iEventGroup].aOpMessage[1].fbAlarm.ipArguments.Clear().AddDInt(stDoor.iIdHMI);
				fbEventHMI(iEventGroup:=GV_Doors.aId[iDoorNumber].iEventGroup,iIdEvent:=1,strEventType:='OpMESSAGE',bEventSet:=TRUE);
			ELSE
				fbEventHMI(iEventGroup:=GV_Doors.aId[iDoorNumber].iEventGroup,iIdEvent:=1,strEventType:='OpMESSAGE',bEventSet:=FALSE);			
			END_IF
			
		END_IF
	
ELSE
	stDoor.bDoorCloseLock:=TRUE; // Door cloe and lock if absent
END_IF

END_FUNCTION_BLOCK

// ---- 07_Cyltronic/03_POUs/01_PRGs/PRG_Cyltronic.TcPOU
PROGRAM PRG_Cyltronic
VAR
	(** INT **)
		iCyltronicLoop : INT := 0 ; // INT use in a FOR Loop
	
	(** FB **)
		fbEventGroupAssignement : FB_Event_Group_Number_Assignement ;
		fbCyltronic : FB_Cyltronic ;
END_VAR

//-----------------------------------------------------------------------------------------
//
//                  				PRG_Cyltronic
//
//					Paramétrage porte(s) Cyltronic + Appel Gestion  			
//-----------------------------------------------------------------------------------------
//
//Auteur: G.GOETZ
//Création: 04.03.2026
//Dernière modification : 04.03.2026 (G.GOETZ)
//       			
//-----------------------------------------------------------------------------------------
//
//     							Liste des modifications  	
//
// 04.03.2026 (G.GOETZ) -> Création		
//-----------------------------------------------------------------------------------------

(** CYLTRONIC : CTC-060-K10-0200-A-IOL -> INTERMEDIATE DOOR **)
	GV_Cyltronic.aId[1].bPresence:=TRUE;
	fbEventGroupAssignement(iEventGroup:=GV_Cyltronic.aId[1].iEventGroup);
	GV_Cyltronic.aId[1].iIdHMI:=1; // Number for events on HMI
	GV_Cyltronic.aId[1].eType:=ENUM_Cyltronic_Type.IOLink; // Cyltronic type
	(* For IO/Link *)
		GV_Cyltronic.aId[1].netID:='10.1.176.55.3.8'; // AmsNetId for IO/Link 10.1.176.55.3.8
		GV_Cyltronic.aId[1].ePort:=E_IolPort.Port1; // Port Number
		//GV_Cyltronic.aId[1].stConfigWrite.MaxSpeedFreePositioning:=150; // Min = 1mm/s - Max = 600mm/s at voltage of 48V
		//GV_Cyltronic.aId[1].stConfigWrite.MaxForceFreePositioning:=120; // Min = 0N - Max = 400N (500N in datasheet)
		//GV_Cyltronic.aId[1].stConfigWrite.MaxAccDec:=2; // Min = 0.01m/s² - Max = 4m/s² (20m/s² in datasheet at voltage of 48V)
		//GV_Cyltronic.aId[1].stConfigWrite.EndPositionIn:=200.0; // mm Depend of the hardware (see datasheet)
		//GV_Cyltronic.aId[1].stConfigWrite.EndPositionOut:=0.0; // mm Depend of the hardware (see datasheet)	
		//GV_Cyltronic.aId[1].stConfigWrite.HomeMode:=CTC_HOME_MODE_ENDSTOPOUT; // Home on In
		(*Limit MaxSpeedFreePositioning*)
			IF GV_Cyltronic.aId[1].stConfigWrite.MaxSpeedFreePositioning<1 THEN
				GV_Cyltronic.aId[1].stConfigWrite.MaxSpeedFreePositioning:=1;
			END_IF
			IF GV_Cyltronic.aId[1].stConfigWrite.MaxSpeedFreePositioning>GV_Cyltronic.aId[1].stConfigDefault.MaxSpeedFreePositioning THEN
				GV_Cyltronic.aId[1].stConfigWrite.MaxSpeedFreePositioning:=GV_Cyltronic.aId[1].stConfigDefault.MaxSpeedFreePositioning;
			END_IF
		(*Limit MaxForceFreePositioning*)
			IF GV_Cyltronic.aId[1].stConfigWrite.MaxForceFreePositioning<0 THEN
				GV_Cyltronic.aId[1].stConfigWrite.MaxSpeedFreePositioning:=0;
			END_IF
			IF GV_Cyltronic.aId[1].stConfigWrite.MaxForceFreePositioning>GV_Cyltronic.aId[1].stConfigDefault.MaxForceFreePositioning THEN
				GV_Cyltronic.aId[1].stConfigWrite.MaxForceFreePositioning:=GV_Cyltronic.aId[1].stConfigDefault.MaxForceFreePositioning;
			END_IF
		(*Limit MaxAccDec*)
			IF GV_Cyltronic.aId[1].stConfigWrite.MaxAccDec<0.01 THEN
				GV_Cyltronic.aId[1].stConfigWrite.MaxAccDec:=0.01;
			END_IF
			IF GV_Cyltronic.aId[1].stConfigWrite.MaxAccDec>GV_Cyltronic.aId[1].stConfigDefault.MaxAccDec THEN
				GV_Cyltronic.aId[1].stConfigWrite.MaxAccDec:=GV_Cyltronic.aId[1].stConfigDefault.MaxAccDec;
			END_IF
		(*Power*)
			IF (GV_General.bSafety AND GV_General.bPower AND (NOT GV_Cyltronic.aId[1].bAlDriveFault)) OR (GV_Cyltronic.aId[1].bPowerEnable AND GV_Cyltronic.aId[1].bHaltExecute AND (NOT GV_Cyltronic.aId[1].bHaltDone))  THEN
				GV_Cyltronic.aId[1].bPowerEnable:=TRUE;
			ELSE
				GV_Cyltronic.aId[1].bPowerEnable:=FALSE;
			END_IF
		(*Halt*)
			GV_Cyltronic.aId[1].bHaltExecute:=(NOT GV_General.bSafety) OR (NOT GV_General.bPower) OR GV_General.bRebootRequest OR GV_General.bShutdownRequest OR (GV_OpMode.eOpMode=ENUM_OpMode.AUTO AND GV_Cycle.bCycleInProgress AND (NOT GV_Cycle.bStartStop)); // Have to halt
		(*Reset*)
			GV_Cyltronic.aId[1].bEventAck:=GV_HMI.bEventAck; // Events Acknowledgement

	(* Work Manual Authorization *)
		IF GV_OpMode.eOpMode=ENUM_OpMode.MANU AND GV_Cyltronic.aId[1].eState=teCTCStep.FB_CTC_READY AND GV_Tool_Magazine.stArm.lrArmPosition<=(GV_Tool_Magazine.stArm.lrArmManipulator+GV_Tool_Magazine.stArm.lrArmPositionTol) (*(GV_Tool_Magazine.stArm.ePositionAxis=ENUM_Position_Axis.Home OR GV_Tool_Magazine.stArm.ePositionAxis=ENUM_Position_Axis.Work1)*) AND ((GV_CNC.stFanucData.stCncMagazine.biAllowedOpenIntermediateDoor AND GV_CNC.bEnable) OR (NOT GV_CNC.bEnable)) AND (NOT GV_Cyltronic.aId[1].bRestPositionCmd) (*AND (NOT GV_Cyltronic.aId[1].bWorkPositionDone)*) THEN
			GV_Cyltronic.aId[1].bAuthorizationManuCyltronicWork:=TRUE;
		ELSE
			GV_Cyltronic.aId[1].bAuthorizationManuCyltronicWork:=FALSE;
			//GV_Cyltronic.aId[1].bWorkPositionCmd:=FALSE;
		END_IF
	(* Work Auto Authorization *)
		IF (GV_OpMode.eOpMode=ENUM_OpMode.AUTO AND GV_Cycle.bStartStop AND GV_Cyltronic.aId[1].eState=teCTCStep.FB_CTC_READY AND (GV_Tool_Magazine.stArm.ePositionAxis=ENUM_Position_Axis.Home OR GV_Tool_Magazine.stArm.ePositionAxis=ENUM_Position_Axis.Work1) AND ((GV_CNC.stFanucData.stCncMagazine.biAllowedOpenIntermediateDoor AND GV_CNC.bEnable) OR (NOT GV_CNC.bEnable)) AND (NOT GV_Cyltronic.aId[1].bRestPositionCmd)) THEN
			GV_Cyltronic.aId[1].bAuthorizationAutoCyltronicWork:=TRUE;
		ELSE
			GV_Cyltronic.aId[1].bAuthorizationAutoCyltronicWork:=FALSE;
			GV_Cycle.bOpenIntermediateDoorRequest:=FALSE;
		END_IF
	(* Work Command *)
		GV_Cyltronic.aId[1].rtWorkPositionCmd(CLK:=GV_Cyltronic.aId[1].bAuthorizationAutoCyltronicWork AND (NOT GV_Cycle.bCloseIntermediateDoorRequest) AND GV_Cycle.bOpenIntermediateDoorRequest);
		IF (GV_Cyltronic.aId[1].rtWorkPositionCmd.Q OR (GV_Cyltronic.aId[1].bAuthorizationManuCyltronicWork AND GV_HMI.stCyltronic.rtButtonMoveWork.Q)) THEN
			GV_Cyltronic.aId[1].bWorkPositionCmd:=TRUE;
		END_IF
		IF GV_Cyltronic.aId[1].bWorkPositionCmd AND (GV_Cyltronic.aId[1].bWorkPositionDone OR GV_HMI.bEventAck) THEN
			GV_Cyltronic.aId[1].bWorkPositionCmd:=FALSE;
		END_IF
		
	(* Rest Manual Authorization *)
		IF GV_OpMode.eOpMode=ENUM_OpMode.MANU AND GV_Cyltronic.aId[1].eState=teCTCStep.FB_CTC_READY AND GV_Tool_Magazine.stArm.lrArmPosition<=(GV_Tool_Magazine.stArm.lrArmManipulator+GV_Tool_Magazine.stArm.lrArmPositionTol) (*(GV_Tool_Magazine.stArm.ePositionAxis=ENUM_Position_Axis.Home OR GV_Tool_Magazine.stArm.ePositionAxis=ENUM_Position_Axis.Work1)*) AND (NOT GV_Cyltronic.aId[1].bWorkPositionCmd) (*AND (NOT GV_Cyltronic.aId[1].bRestPositionDone)*) THEN
			GV_Cyltronic.aId[1].bAuthorizationManuCyltronicRest:=TRUE;
		ELSE
			GV_Cyltronic.aId[1].bAuthorizationManuCyltronicRest:=FALSE;
			//GV_Cyltronic.aId[1].bRestPositionCmd:=FALSE;
		END_IF
	(* Rest Auto Authorization *)
		IF (GV_OpMode.eOpMode=ENUM_OpMode.AUTO AND GV_Cycle.bStartStop AND GV_Cyltronic.aId[1].eState=teCTCStep.FB_CTC_READY AND (GV_Tool_Magazine.stArm.ePositionAxis=ENUM_Position_Axis.Home OR GV_Tool_Magazine.stArm.ePositionAxis=ENUM_Position_Axis.Work1) AND (NOT GV_Cyltronic.aId[1].bWorkPositionCmd)) THEN
			GV_Cyltronic.aId[1].bAuthorizationAutoCyltronicRest:=TRUE;
		ELSE
			GV_Cyltronic.aId[1].bAuthorizationAutoCyltronicRest:=FALSE;
			GV_Cycle.bCloseIntermediateDoorRequest:=FALSE;
		END_IF
	(* Rest Command *)
		GV_Cyltronic.aId[1].rtRestPositionCmd(CLK:=GV_Cyltronic.aId[1].bAuthorizationAutoCyltronicRest AND GV_Cycle.bCloseIntermediateDoorRequest AND (NOT GV_Cycle.bOpenIntermediateDoorRequest));
		IF (GV_Cyltronic.aId[1].rtRestPositionCmd.Q OR (GV_Cyltronic.aId[1].bAuthorizationManuCyltronicRest AND GV_HMI.stCyltronic.rtButtonMoveRest.Q)) THEN
			GV_Cyltronic.aId[1].bRestPositionCmd:=TRUE;
		END_IF
		IF GV_Cyltronic.aId[1].bRestPositionCmd AND (GV_Cyltronic.aId[1].bRestPositionDone OR GV_HMI.bEventAck) THEN
			GV_Cyltronic.aId[1].bRestPositionCmd:=FALSE;
		END_IF
		
		
(** OTHER CYLTRONIC **)
//...

(** FB **)
	FOR iCyltronicLoop:=1 TO GV_Cyltronic.iMaxCyltronic DO
		fbCyltronic(iCyltroNumber:=iCyltronicLoop,StCyltronic:=GV_Cyltronic.aId[iCyltronicLoop]); // Cyltronic function block
	END_FOR

END_PROGRAM

// ---- 07_Cyltronic/03_POUs/02_FBs/FB_Cyltronic.TcPOU
FUNCTION_BLOCK FB_Cyltronic
VAR_INPUT
	(** INT **)
		iCyltroNumber : INT ; // Number of the cyltronic
END_VAR
VAR_OUTPUT
END_VAR
VAR_IN_OUT
	(** ST **)
		stCyltronic : ST_Cyltronic ;
END_VAR
VAR
	(** FLAG **)
		(*fbCTC*)
			bCTCDone : BOOL ; // fbCTCPlcOpen is Done
			bCTCBusy : BOOL ; // fbCTCPlcOpen is Busy
			bCTCWarning : BOOL ; // fbCTCPlcOpen Warning
			bCTCError : BOOL ; // fbCTCPlcOpen Error	
		bTeachStart : BOOL ;
		bHomeStart : BOOL ;
		bHalt : BOOL ;

	(** FB **)
		fbInitEvents : FB_Init_Events ;
		fbEventHMI : FB_Event_HMI ;
	
		fbCTCBasic : FB_CTC_Basic ;
		fbCTCReadConfig : FB_CTC_ReadWriteConfig ;
		fbCTCWriteConfig : FB_CTC_ReadWriteConfig ;
		fbCTCGetDeviceStatus : FB_CTC_GetDeviceStatus ;
		fbCTCPlcOpen : FB_CTC_PlcOpen ;
		
bEssai : BOOL ;
		
END_VAR

//-----------------------------------------------------------------------------------------
//
//                  				FB_Cyltronic
//
//								Gestion Cyltronic 			
//-----------------------------------------------------------------------------------------
//
//Auteur: G.GOETZ
//Création: 04.03.2026
//Dernière modification : 04.03.2026 (G.GOETZ)
//       			
//-----------------------------------------------------------------------------------------
//
//     							Liste des modifications  	
//
// 04.03.2026 (G.GOETZ) -> Création	
//-----------------------------------------------------------------------------------------

IF stCyltronic.bPresence THEN
		
	(** EVENTS **)
		IF GV_General.bFirstCycleTask OR GV_General.bFirstCycleSimu THEN
			GV_Events.aEventGroup[GV_Cyltronic.aId[iCyltroNumber].iEventGroup].aAlarm[1].fbAlarm.CreateEx(TC_Events.CyltronicAlarms.Alarm1,TRUE,0);
			GV_Events.aEventGroup[GV_Cyltronic.aId[iCyltroNumber].iEventGroup].aOpMessage[1].fbAlarm.CreateEx(TC_Events.CyltronicOpMessages.Message1,TRUE,0);	
			fbInitEvents(iEventGroup:=GV_Cyltronic.aId[iCyltroNumber].iEventGroup,strEventType:='ALARM',strEventGuid:='B84E62CB-48E4-46DB-ADFD-2D2E7A2978F6',tcEventSeverity:=2);
			fbInitEvents(iEventGroup:=GV_Cyltronic.aId[iCyltroNumber].iEventGroup,strEventType:='OpMESSAGE',strEventGuid:='6E644DA8-210C-419D-A327-FA38AE35A6A6',tcEventSeverity:=1);
		END_IF
			
	(** ALARMS **)
		(* Drive fault *)
			(*Reset fault*)
				IF stCyltronic.bEventAck THEN
					stCyltronic.bAlDriveFault:=FALSE;
				END_IF
			(*Set fault*)
				IF stCyltronic.eState=teCTCStep.FB_CTC_ERROR THEN
					stCyltronic.bAlDriveFault:=TRUE;
				END_IF
			(*Alarm 1 = Drive in fault*)
				IF stCyltronic.bAlDriveFault THEN
					GV_Events.aEventGroup[GV_Cyltronic.aId[iCyltroNumber].iEventGroup].aAlarm[1].fbAlarm.ipArguments.Clear().AddDInt(stCyltronic.iIdHMI);
					fbEventHMI(iEventGroup:=stCyltronic.iEventGroup,iIdEvent:=1,strEventType:='ALARM',bEventSet:=TRUE);
				ELSE
					fbEventHMI(iEventGroup:=stCyltronic.iEventGroup,iIdEvent:=1,strEventType:='ALARM',bEventSet:=FALSE);			
				END_IF
				
	(** MESSAGES **)

	(** CYLTRONIC TYPES MANAGEMENT **)
	
	(* 1 DiDo Technology *)
		//IF stCyltronic.eType=ENUM_Cyltronic_Type.DiDo THEN
			
		//END_IF
	
	(* 2 IO/Link Technology *)	
		IF stCyltronic.eType=ENUM_Cyltronic_Type.IOLink THEN
			(* Configuration Read (acyclic) *)
				fbCTCReadConfig(
								// IN
								AmsNetid:=stCyltronic.netID,
								IolPort:=stCyltronic.ePort,
								Read:=GV_General.bIsBlinking1s,
								Write:=FALSE,
								// IN_OUT
								pstConfiguration:=stCyltronic.stConfigRead,
								// OUT
								Busy=>,
								Done=>,
								AtLeastOneParameterFailed=>,
							   );
							   
			(* Configuration Write (acyclic) *)
				IF (stCyltronic.stConfigRead.MaxSpeedFreePositioning<>stCyltronic.stConfigWrite.MaxSpeedFreePositioning OR 
					stCyltronic.stConfigRead.MaxForceFreePositioning<>stCyltronic.stConfigWrite.MaxForceFreePositioning OR
					stCyltronic.stConfigRead.MaxAccDec<>stCyltronic.stConfigWrite.MaxAccDec OR
					stCyltronic.stConfigRead.HomeMode<>stCyltronic.stConfigWrite.HomeMode OR
					stCyltronic.stConfigRead.EndPositionOut<>stCyltronic.stConfigWrite.EndPositionOut OR
					stCyltronic.stConfigRead.EndPositionIn<>stCyltronic.stConfigWrite.EndPositionIn) 
					AND (NOT fbCTCReadConfig.Busy) THEN
					stCyltronic.bStartWriteConfig:=TRUE;
				ELSE
					stCyltronic.bStartWriteConfig:=FALSE;
				END_IF
			
				fbCTCWriteConfig(
								// IN
								AmsNetid:=stCyltronic.netID,
								IolPort:=stCyltronic.ePort,
								Read:=FALSE,
								Write:=FALSE,//stCyltronic.bStartWriteConfig,
								// IN_OUT
								pstConfiguration:=stCyltronic.stConfigWrite,
								// OUT
								Busy=>,
								Done=>,
								AtLeastOneParameterFailed=>,
							   );
							   
			(* Status (acyclic) *)
				fbCTCGetDeviceStatus(
									// IN
									AmsNetid:=stCyltronic.netID,
									IolPort:=stCyltronic.ePort,
									GetStatus:=GV_General.bIsBlinking1s AND (NOT fbCTCGetDeviceStatus.Busy),
									// OUT
									stDeviceStatus=>stCyltronic.stStatus,
									Busy=>,
									Done=>,
									Failed=>,
									);

			(* Exchange *)
// 				fbCTCBasic(
// 						   // IN
// 						   ProcessDataInRaw:=stCyltronic.aProcessDataInRaw,
// 						   MotionMode:=,
// 						   
// 						   // OUT
// 						   ProcessDataOutRaw=>stCyltronic.aProcessDataOutRaw,
// 						   State=>stCyltronic.eState,
// 						   
// 						   
// 						   );
				stCyltronic.stParameters.TargetPosition:=stCyltronic.stConfigRead.EndPositionOut-4.136;//181.7;
				stCyltronic.stParameters.TargetForce:=200;
				fbCTCPlcOpen(
							// IN
							ProcessDataInRaw:=stCyltronic.aProcessDataInRaw,
							Enable:=stCyltronic.bPresence,
							Power:=stCyltronic.bPowerEnable,
							Teach:=bTeachStart,
							Home:=bHomeStart,
							MoveIn:=stCyltronic.bWorkPositionCmd,// AND fbCTCPlcOpen.Homed,
							MoveOut:=,//stCyltronic.bRestPositionCmd,// AND fbCTCPlcOpen.Homed,
							MoveAbsolute:=stCyltronic.bRestPositionCmd,
							MoveContinuous:=,
							Halt:=stCyltronic.bHaltExecute OR bHalt,
							Reset:=stCyltronic.bEventAck,
							BrakeMode:=,
							BrakeDelay:=,
							stParameters:=stCyltronic.stParameters,
							stConfiguration:=stCyltronic.stConfigRead, // Not for write the config but to compare
							// OUT
							ProcessDataOutRaw=>stCyltronic.aProcessDataOutRaw,
							State=>stCyltronic.eState,
							ControllerOn=>,
							ActualPosition=>,
							ActualVelocity=>,
							ActualForce=>,
							Homed=>,
							Busy=>bCTCBusy,
							Done=>bCTCDone,
							Warning=>bCTCWarning,
							WarningID=>,
							Error=>bCTCError,
							ReleaseBrake=>,
							stProcessDataIn=>stCyltronic.stProcessDataIn,
							stProcessDataOut=>stCyltronic.stProcessDataOut,
							);
							
			(* Work Done *)
				IF stCyltronic.bWorkPositionCmd AND stCyltronic.stProcessDataIn.stStatusBits.LimitSwitchIn AND stCyltronic.stProcessDataIn.stStatusBits.MotionCommandCompleted AND (NOT bCTCBusy) THEN
					stCyltronic.bWorkPositionDone:=TRUE;
					stCyltronic.bRestPositionDone:=FALSE;
				END_IF
			(* Rest Done *)
				IF stCyltronic.bRestPositionCmd AND (*stCyltronic.stProcessDataIn.stStatusBits.LimitSwitchOut AND*) stCyltronic.stProcessDataIn.stStatusBits.MotionCommandCompleted AND (NOT bCTCBusy) THEN
					stCyltronic.bWorkPositionDone:=FALSE;
					stCyltronic.bRestPositionDone:=TRUE;
				END_IF
			(* Halt Done *)
				IF stCyltronic.bHaltExecute AND (NOT bCTCBusy) AND bCTCDone THEN
					stCyltronic.bHaltDone:=TRUE;
					stCyltronic.bWorkPositionDone:=FALSE;
					stCyltronic.bRestPositionDone:=FALSE;
				ELSE
					stCyltronic.bHaltDone:=FALSE;
				END_IF
		END_IF
	
//ELSE

END_IF

END_FUNCTION_BLOCK

// ---- 07_Cyltronic/03_POUs/02_FBs/FB_CTC_Basic.TcPOU
FUNCTION_BLOCK FB_CTC_Basic
VAR_INPUT
	ProcessDataInRaw 	:ARRAY[0..13] OF BYTE;
	MotionMode 			:USINT;
	TargetPosition 		:REAL;
	Override1 			:USINT;
	Override2 			:USINT;
	Override3 			:USINT;
END_VAR
VAR_OUTPUT
	ProcessDataOutRaw 	:ARRAY[0..7] OF BYTE;
	State 				:USINT;
	StatusBits 			:tstCTCStatusBits;
	ActualPosition 		:REAL;
	ActualSpeed 		:REAL;
	ActualForce 		:REAL;
END_VAR
VAR
	stProcessDataIn 	:tstCTCProcessDataIn;
	stProcessDataOut 	:tstCTCProcessDataOut;
	unionContainer		:tuReal;
END_VAR

(*
	FB_CTC_Basic V3.0
	Cyltronic AG, September 2024

	Function Block that handles process data in raw octet form of Cyltronic devices
	and provides according process data structure
*)
// =================================================================================
// === PROCESS DATA INPUTS =========================================================
// =================================================================================
// Status = Byte 0
stProcessDataIn.State := BYTE_TO_USINT(ProcessDataInRaw[0]);
// StatusBits = Byte 1
stProcessDataIn.stStatusBits.TrackingErrorToleranceExceeded	:= ProcessDataInRaw[1].7;
stProcessDataIn.stStatusBits.WarningActive 					:= ProcessDataInRaw[1].6;
stProcessDataIn.stStatusBits.MotionCommandCompleted 		:= ProcessDataInRaw[1].5;
stProcessDataIn.stStatusBits.MotionModeActive 				:= ProcessDataInRaw[1].4;
stProcessDataIn.stStatusBits.LimitSwitchIn 					:= ProcessDataInRaw[1].3;
stProcessDataIn.stStatusBits.LimitSwitchOut 				:= ProcessDataInRaw[1].2;
stProcessDataIn.stStatusBits.Homed 							:= ProcessDataInRaw[1].1;
stProcessDataIn.stStatusBits.Ready 							:= ProcessDataInRaw[1].0;
// Actual Position = Bytes 2-5
unionContainer.aBytes[0] := ProcessDataInRaw[5];
unionContainer.aBytes[1] := ProcessDataInRaw[4];
unionContainer.aBytes[2] := ProcessDataInRaw[3];
unionContainer.aBytes[3] := ProcessDataInRaw[2];
stProcessDataIn.ActualPosition := unionContainer.rReal;
// Actual Speed = Bytes 6-9
unionContainer.aBytes[0] := ProcessDataInRaw[9];
unionContainer.aBytes[1] := ProcessDataInRaw[8];
unionContainer.aBytes[2] := ProcessDataInRaw[7];
unionContainer.aBytes[3] := ProcessDataInRaw[6];
stProcessDataIn.ActualSpeed := unionContainer.rReal;
// Actual Force = Bytes 10-13
unionContainer.aBytes[0] := ProcessDataInRaw[13];
unionContainer.aBytes[1] := ProcessDataInRaw[12];
unionContainer.aBytes[2] := ProcessDataInRaw[11];
unionContainer.aBytes[3] := ProcessDataInRaw[10];
stProcessDataIn.ActualForce := unionContainer.rReal;

// =================================================================================
// === Distribute ==================================================================
// =================================================================================
// Inputs --> CTC to PLC
State 			:= stProcessDataIn.State;
StatusBits 		:= stProcessDataIn.stStatusBits;
ActualPosition 	:= stProcessDataIn.ActualPosition;
ActualSpeed 	:= stProcessDataIn.ActualSpeed;
ActualForce 	:= stProcessDataIn.ActualForce;

// Outputs --> PLC to CTC
stProcessDataOut.MotionMode 	:= MotionMode;
stProcessDataOut.TargetPosition := TargetPosition;
stProcessDataOut.Override1 		:= Override1;
stProcessDataOut.Override2 		:= Override2;
stProcessDataOut.Override3 		:= Override3;

// =================================================================================
// === PD OUTPUTS ==================================================================
// =================================================================================
// Motion Mode
ProcessDataOutRaw[0] := USINT_TO_BYTE(stProcessDataOut.MotionMode);
// Set Position
unionContainer.rReal := stProcessDataOut.TargetPosition;
ProcessDataOutRaw[1] := unionContainer.aBytes[3];
ProcessDataOutRaw[2] := unionContainer.aBytes[2];
ProcessDataOutRaw[3] := unionContainer.aBytes[1];
ProcessDataOutRaw[4] := unionContainer.aBytes[0];
// Overrides 1-3
ProcessDataOutRaw[5] := USINT_TO_BYTE(stProcessDataOut.Override1);
ProcessDataOutRaw[6] := USINT_TO_BYTE(stProcessDataOut.Override2);
ProcessDataOutRaw[7] := USINT_TO_BYTE(stProcessDataOut.Override3);

END_FUNCTION_BLOCK

// ---- 07_Cyltronic/03_POUs/02_FBs/FB_CTC_ReadWriteConfig.TcPOU
FUNCTION_BLOCK FB_CTC_ReadWriteConfig
VAR_INPUT
	AmsNetid 	:T_AmsNetid;
	IolPort		:E_IolPort;
	Read 		:BOOL;
	Write 		:BOOL;
END_VAR
VAR_OUTPUT
	Busy 		:BOOL;
	Done 		:BOOL;
	AtLeastOneParameterFailed :BOOL;
END_VAR
VAR_IN_OUT
	pstConfiguration :tstCTCConfiguration;	
END_VAR

VAR
	FB_IolRead_0 		:FB_IolRead;
	FB_IolWrite_0 		:FB_IolWrite;
	bInit 				:BOOL := FALSE;
	eStep 				:teCTCConfigStep;
	aCTCConfigVariables :ARRAY[0..NUMBER_OF_PARAMETERS] OF tstCTCConfigVariable;
	R_TRIG_Read 		:R_TRIG;
	R_TRIG_Write 		:R_TRIG;
	unionContainer		:tuReal;
	tonTimeout 			:TON;
	iParameterIndex 	:USINT;
	bufferArray			:ARRAY[0..3] OF BYTE;
END_VAR
VAR CONSTANT
	NUMBER_OF_PARAMETERS	:USINT := 6; (*because its and index, its actuall the number of parameters - 1*)
	CTC_DATATYPE_REAL		:USINT := 0;
	CTC_DATATYPE_USINT		:USINT := 1;
	
END_VAR

(*
	FB_CTC_ReadWriteConfig V2.0
	Cyltronic AG, June 2024

	Function Block that reads and writes stConfiguration object used
	in FB_CTC_PlcOpen

	Intended as example function block for reading/writing acyclic data
*)

FB_IolRead_0.sNetId := AmsNetid;
FB_IolRead_0.nIolPort := IolPort;

FB_IolWrite_0.sNetId := AmsNetid;
FB_IolWrite_0.nIolPort := IolPort;

IF(bInit = FALSE)THEN
	bInit := TRUE;	
	
	aCTCConfigVariables[0].Name := 'MaxSpeedFreePositioning';
	aCTCConfigVariables[0].Index := 66;
	aCTCConfigVariables[0].Subindex := 0;
	aCTCConfigVariables[0].DataType := CTC_DATATYPE_REAL;
	aCTCConfigVariables[0].ValueIfReal := 0;
	
	aCTCConfigVariables[1].Name := 'MaxForceFreePositioning';
	aCTCConfigVariables[1].Index := 84;
	aCTCConfigVariables[1].Subindex := 0;
	aCTCConfigVariables[1].DataType := CTC_DATATYPE_REAL;
	aCTCConfigVariables[1].ValueIfReal := 0;
	
	aCTCConfigVariables[2].Name := 'MaxAcceleration';
	aCTCConfigVariables[2].Index := 68;
	aCTCConfigVariables[2].Subindex := 0;
	aCTCConfigVariables[2].DataType := CTC_DATATYPE_REAL;
	aCTCConfigVariables[2].ValueIfReal := 0;
			
	aCTCConfigVariables[3].Name := 'MaxDeceleration';
	aCTCConfigVariables[3].Index := 69;
	aCTCConfigVariables[3].Subindex := 0;
	aCTCConfigVariables[3].DataType := CTC_DATATYPE_REAL;
	aCTCConfigVariables[3].ValueIfReal := 0;
	
	aCTCConfigVariables[4].Name := 'EndPositionIn';
	aCTCConfigVariables[4].Index := 76;
	aCTCConfigVariables[4].Subindex := 0;
	aCTCConfigVariables[4].DataType := CTC_DATATYPE_REAL;
	aCTCConfigVariables[4].ValueIfReal := 0;
	
	aCTCConfigVariables[5].Name := 'EndPositionOut';
	aCTCConfigVariables[5].Index := 75;
	aCTCConfigVariables[5].Subindex := 0;
	aCTCConfigVariables[5].DataType := CTC_DATATYPE_REAL;
	aCTCConfigVariables[5].ValueIfReal := 0;
	
	aCTCConfigVariables[6].Name := 'HomeMode';
	aCTCConfigVariables[6].Index := 261;
	aCTCConfigVariables[6].Subindex := 0;
	aCTCConfigVariables[6].DataType := CTC_DATATYPE_USINT;
	aCTCConfigVariables[6].ValueIfUSINT := 0;
	
	Busy := FALSE;
	Done := FALSE;
	AtLeastOneParameterFailed := FALSE;
	
END_IF;

CASE eStep OF
	// ====================================================
	// === P_IDLE =========================================
	// ====================================================
	CTC_CONFIG_IDLE:

		FB_IolRead_0.bExecute := FALSE;
		FB_IolWrite_0.bExecute := FALSE;
		tonTimeout.IN := FALSE;
	
		R_TRIG_Read.CLK := Read;
		R_TRIG_Write.CLK := Write;
		
		IF(R_TRIG_Read.Q)THEN
			iParameterIndex := 0;
			eStep := CTC_CONFIG_READ_START;
		ELSIF(R_TRIG_Write.Q)THEN
			iParameterIndex := 0;
			eStep := CTC_CONFIG_WRITE_PREPARE;
		END_IF
			
	// ======================================================================================================
	// === CTC_CONFIG_READ_START ============================================================================
	// ======================================================================================================
	CTC_CONFIG_READ_START:
			
		Busy := TRUE;
		Done := FALSE;
		AtLeastOneParameterFailed := FALSE;
			
		FB_IolRead_0.pDSTBuf	:= ADR(bufferArray);
		IF(aCTCConfigVariables[iParameterIndex].DataType = CTC_DATATYPE_REAL)THEN
			FB_IolRead_0.cbBufLen	:= 4;
		ELSIF(aCTCConfigVariables[iParameterIndex].DataType = CTC_DATATYPE_USINT)THEN
			FB_IolRead_0.cbBufLen	:= 1;
		END_IF
		FB_IolRead_0.nIndex 	:= aCTCConfigVariables[iParameterIndex].Index;
		FB_IolRead_0.nSubindex 	:= aCTCConfigVariables[iParameterIndex].Subindex;
		FB_IolRead_0.bExecute	:= TRUE;
				
		tonTimeout.IN := FALSE;
			
		eStep := CTC_CONFIG_READ_WAIT;
	
	// ====================================================
	// === CTC_CONFIG_READ_WAIT ===========================
	// ====================================================
	CTC_CONFIG_READ_WAIT:
			
		tonTimeout.IN := TRUE;

		IF((FB_IolRead_0.bDone) OR tonTimeout.Q)THEN
			AtLeastOneParameterFailed := AtLeastOneParameterFailed OR tonTimeout.Q;
			FB_IolRead_0.bExecute := FALSE;
				
			// process data, depending on datatype
			IF (aCTCConfigVariables[iParameterIndex].DataType = CTC_DATATYPE_REAL) THEN
                unionContainer.aBytes[0] := bufferArray[3];
				unionContainer.aBytes[1] := bufferArray[2];
				unionContainer.aBytes[2] := bufferArray[1];
				unionContainer.aBytes[3] := bufferArray[0];
                aCTCConfigVariables[iParameterIndex].ValueIfReal := unionContainer.rReal;
            ELSIF(aCTCConfigVariables[iParameterIndex].Datatype = CTC_DATATYPE_USINT)THEN
                aCTCConfigVariables[iParameterIndex].ValueIfUSint := BYTE_TO_USINT(bufferArray[0]);
            END_IF;
				
			// next parameter, or finished
			iParameterIndex := iParameterIndex + 1;
			IF(iParameterIndex <= NUMBER_OF_PARAMETERS)THEN
				eStep := CTC_CONFIG_READ_START;
			ELSE
				eStep := CTC_CONFIG_READ_FINISH;
			END_IF	
		
		END_IF
			
	// ====================================================
	// === CTC_CONFIG_READ_FINISH =========================
	// ====================================================
	CTC_CONFIG_READ_FINISH:
			
		pstConfiguration.MaxSpeedFreePositioning := aCTCConfigVariables[0].ValueIfReal;
		pstConfiguration.MaxForceFreePositioning := aCTCConfigVariables[1].ValueIfReal;
		pstConfiguration.MaxAccDec := aCTCConfigVariables[2].ValueIfReal;
		pstConfiguration.EndPositionIn := aCTCConfigVariables[4].ValueIfReal;
		pstConfiguration.EndPositionOut := aCTCConfigVariables[5].ValueIfReal;
		pstConfiguration.HomeMode := aCTCConfigVariables[6].ValueIfUSINT;
		
		Busy := FALSE;
		Done := TRUE;
		
		eStep := CTC_CONFIG_IDLE;
		
	// ======================================================================================================
	// === CTC_CONFIG_WRITE_PREPARE =========================================================================
	// ======================================================================================================
	CTC_CONFIG_WRITE_PREPARE:

		Busy := TRUE;
		Done := FALSE;
		AtLeastOneParameterFailed := FALSE;
		
		aCTCConfigVariables[0].ValueIfReal 	:= pstConfiguration.MaxSpeedFreePositioning;
		aCTCConfigVariables[1].ValueIfReal 	:= pstConfiguration.MaxForceFreePositioning;
		aCTCConfigVariables[2].ValueIfReal 	:= pstConfiguration.MaxAccDec;
		aCTCConfigVariables[3].ValueIfReal 	:= pstConfiguration.MaxAccDec;
		aCTCConfigVariables[4].ValueIfReal 	:= pstConfiguration.EndPositionIn;
		aCTCConfigVariables[5].ValueIfReal 	:= pstConfiguration.EndPositionOut;
		aCTCConfigVariables[6].ValueIfUSINT := DINT_TO_USINT(pstConfiguration.HomeMode);
			
		FB_IolWrite_0.bExecute := FALSE;
			
		eStep := CTC_CONFIG_WRITE_START;
			
	// ====================================================
	// === CTC_CONFIG_WRITE_START =========================
	// ====================================================
	CTC_CONFIG_WRITE_START:
			
		// process data, depending on datatype
	
		IF(aCTCConfigVariables[iParameterIndex].DataType = CTC_DATATYPE_REAL)THEN
			unionContainer.rReal := aCTCConfigVariables[iParameterIndex].ValueIfReal;
			bufferArray[0] := 	unionContainer.aBytes[3];
			bufferArray[1] := 	unionContainer.aBytes[2];
			bufferArray[2] := 	unionContainer.aBytes[1];
			bufferArray[3] := 	unionContainer.aBytes[0];
			FB_IolWrite_0.cbBufLen 	:= 4;
		ELSIF(aCTCConfigVariables[iParameterIndex].DataType = CTC_DATATYPE_USINT)THEN
			bufferArray[0] := aCTCConfigVariables[iParameterIndex].ValueIfUSINT;
			FB_IolWrite_0.cbBufLen := 1;
		END_IF
			
		FB_IolWrite_0.pSRCBuf	:= ADR(bufferArray);
		FB_IolWrite_0.nIndex 	:= aCTCConfigVariables[iParameterIndex].Index;
		FB_IolWrite_0.nSubindex := aCTCConfigVariables[iParameterIndex].Subindex;
		FB_IolWrite_0.bExecute 	:= TRUE;
		
		tonTimeout.IN := FALSE;
		
		eStep := CTC_CONFIG_WRITE_WAIT;
		
	// ====================================================
	// === CTC_CONFIG_WRITE_WAIT ==========================
	// ====================================================
	CTC_CONFIG_WRITE_WAIT:
			
		tonTimeout.IN := TRUE;
	
		IF((FB_IolWrite_0.bDone = TRUE) OR tonTimeout.Q)THEN
			AtLeastOneParameterFailed := AtLeastOneParameterFailed OR tonTimeout.Q;
			FB_IolWrite_0.bExecute := FALSE;
			
			iParameterIndex := iParameterIndex + 1;
			IF(iParameterIndex <= NUMBER_OF_PARAMETERS)THEN
				eStep := CTC_CONFIG_WRITE_START;
			ELSE
				Busy := FALSE;
				Done := TRUE;
				eStep := CTC_CONFIG_IDLE;
			END_IF	
			
		END_IF
		
	ELSE
		eStep := CTC_CONFIG_IDLE;
			
END_CASE;
	
//call FBs
R_TRIG_Read();
R_TRIG_Write();
tonTimeout(PT := T#2S);
FB_IolRead_0();
FB_IolWrite_0();

END_FUNCTION_BLOCK

// ---- 07_Cyltronic/03_POUs/02_FBs/FB_CTC_GetDeviceStatus.TcPOU
FUNCTION_BLOCK FB_CTC_GetDeviceStatus
VAR_INPUT
	AmsNetid 		:T_AmsNetid;
	IolPort			:E_IolPort;
	GetStatus		:BOOL;
END_VAR
VAR_OUTPUT
	stDeviceStatus	:tstCTCDeviceStatus;
	Busy 			:BOOL;
	Done 			:BOOL;
	Failed 			:BOOL;
END_VAR
VAR
	FB_IolRead_0 		:FB_IolRead;
	bInit 				:BOOL := FALSE;
	eStep 				:teCTCGDSStep;
	bufferArray			:ARRAY[0..56] OF BYTE;	// must be 57 bytes long: 19 Events with each 3 bytes
	tonTimeout 			:TON;
	R_TRIG_GetStatus	:R_TRIG;
	iEventIndex			:USINT;
	temp_word1			:WORD;
	temp_word2			:WORD;
	temp_word3			:WORD;
END_VAR
VAR CONSTANT
	INDEX_DEVICE_STATUS				:USINT := 36;
	INDEX_DETAILED_DEVICE_STATUS	:USINT := 37;
	NUMBER_OF_EVENTS				:USINT := 4;	// because its an index, its number of events - 1
END_VAR

(*
	FB_CTC_GetDeviceStatus V2.0
	Cyltronic AG, June 2024

	Function Block that reads Index 36 and 37 to provide detailed information
	of current IO-Link events 
*)

FB_IolRead_0.sNetId := AmsNetid;
FB_IolRead_0.nIolPort := IolPort;

IF(bInit = FALSE)THEN
	bInit := TRUE;	

	Busy 	:= FALSE;
	Done 	:= FALSE;
	Failed 	:= FALSE;
END_IF;

CASE eStep OF
        // ====================================================
        // === #CTC_GDS_IDLE ==================================
        // ====================================================
    CTC_GDS_IDLE:
        
		FB_IolRead_0.bExecute := FALSE;
		tonTimeout.IN := FALSE;
	
		R_TRIG_GetStatus.CLK := GetStatus;
		
		IF(R_TRIG_GetStatus.Q)THEN
			iEventIndex := 0;
			eStep := CTC_GDS_READ_STATUS_START;
		END_IF
        
        // ====================================================
        // === #CTC_GDS_READ_STATUS_START =====================
        // ====================================================
    CTC_GDS_READ_STATUS_START:
        
        Busy := TRUE;
        Done := FALSE;
        Failed := FALSE;
        
		FB_IolRead_0.pDSTBuf	:= ADR(bufferArray);
		FB_IolRead_0.cbBufLen	:= 1;
		FB_IolRead_0.nIndex 	:= INDEX_DEVICE_STATUS;
		FB_IolRead_0.nSubindex 	:= 0;
		FB_IolRead_0.bExecute	:= TRUE;
        
        tonTimeout.IN := FALSE;
        
        eStep := CTC_GDS_READ_STATUS_WAIT;
        
        // ====================================================
        // === #CTC_GDS_READ_STATUS_WAIT ======================
        // ====================================================
    CTC_GDS_READ_STATUS_WAIT:
        
        tonTimeout.IN := TRUE;
        
        IF ((FB_IolRead_0.bDone = TRUE) OR tonTimeout.Q) THEN
            Failed := Failed OR tonTimeout.Q;
            FB_IolRead_0.bExecute := FALSE;
            
            // process data: Device Status, Index 36, is the first byte
            stDeviceStatus.DeviceStatus := BYTE_TO_INT(bufferArray[0]);
            
            eStep := CTC_GDS_READ_DETSTAT_START;
            
        END_IF;
        
        // ====================================================
        // === CTC_CONFIG_READ_FINISH =========================
        // ====================================================
    CTC_GDS_READ_DETSTAT_START:
        
		FB_IolRead_0.pDSTBuf	:= ADR(bufferArray);
		FB_IolRead_0.cbBufLen	:= 57;
		FB_IolRead_0.nIndex 	:= INDEX_DETAILED_DEVICE_STATUS;
		FB_IolRead_0.nSubindex 	:= 0;
		FB_IolRead_0.bExecute	:= TRUE;
        
        tonTimeout.IN := FALSE;
        
        iEventIndex := 0;
        
        eStep := CTC_GDS_READ_DETSTAT_WAIT;
        
        // ====================================================
        // === CTC_GDS_READ_DETAILED_STATUS_WAIT ==============
        // ====================================================
    CTC_GDS_READ_DETSTAT_WAIT:
        
        tonTimeout.IN := TRUE;
        
        IF ((FB_IolRead_0.bDone = TRUE) OR tonTimeout.Q) THEN
            Failed := Failed OR tonTimeout.Q;
            FB_IolRead_0.bExecute := FALSE;
            
            // process data: Detailed Device Status, Index 37, is the current eventqueue
            // --> 1 byte qulifier, 2 bytes event identifier, then repeat for the next event. We extract the first 5
            FOR iEventIndex := 0 TO NUMBER_OF_EVENTS BY 1 DO
                
                stDeviceStatus.Events[iEventIndex].Qualifier := BYTE_TO_USINT(bufferArray[iEventIndex*3]);
                temp_word1 := BYTE_TO_WORD(bufferArray[iEventIndex*3+2]);
				temp_word2 := BYTE_TO_WORD(bufferArray[iEventIndex*3+1]);
				temp_word3 := temp_word1 OR SHL(temp_word2,8);
				stDeviceStatus.Events[iEventIndex].Event := WORD_TO_INT(temp_word3);
           
            END_FOR;
            
            eStep := CTC_GDS_IDLE;
            Busy := FALSE;
            Done := TRUE;
            
        END_IF;
        
    ELSE
        eStep := CTC_GDS_IDLE;
        
END_CASE;
	
//call FBs
R_TRIG_GetStatus();
tonTimeout(PT := T#2S);
FB_IolRead_0();

END_FUNCTION_BLOCK

// ---- 07_Cyltronic/03_POUs/02_FBs/FB_CTC_PlcOpen.TcPOU
FUNCTION_BLOCK FB_CTC_PlcOpen
VAR_INPUT
	ProcessDataInRaw 	:ARRAY[0..13] OF BYTE;
	Enable				:BOOL;
	Power				:BOOL;
	Teach				:BOOL;
	Home				:BOOL;
	MoveIn				:BOOL;
	MoveOut				:BOOL;
	MoveAbsolute		:BOOL;
	MoveContinuous		:BOOL;
	Halt				:BOOL;
	Reset				:BOOL;
	BrakeMode			:teCTCBrakeMode := CTC_BRAKE_MODE_OFF;
	BrakeDelay			:UINT := 100;
	stParameters		:tstCTCParameters;
	stConfiguration		:tstCTCConfiguration;
END_VAR
VAR_OUTPUT
	ProcessDataOutRaw 	:ARRAY[0..7] OF BYTE;
	State				:teCTCStep;
	ControllerOn		:BOOL;
	ActualPosition		:REAL;
	ActualVelocity		:REAL;
	ActualForce			:REAL;
	Homed				:BOOL;
	Busy				:BOOL;
	Done				:BOOL;
	Warning				:BOOL;
	WarningID			:teCTCWarningID;
	Error				:BOOL;
	ReleaseBrake		:BOOL;
	stProcessDataIn		:tstCTCProcessDataIn;
	stProcessDataOut	:tstCTCProcessDataOut;
END_VAR
VAR
	bInit				:BOOL := FALSE;
	eStep				:teCTCStep;
	unionContainer		:tuReal;
	stInternalCommands	:tstCTCInternalCommands;
	R_TRIG_Array		:ARRAY[0..6] OF R_TRIG;
	R_TRIG_Reset		:R_TRIG;
	iIntermediateStep 	:USINT;
	TON_MMComplete		:TON;
	TON_Reset			:TON;
	TON_Brake			:TON;
	bSetpointError 		:BOOL;
	bHomeTeachFailed	:BOOL;
END_VAR
VAR CONSTANT
	FREE_POS_TOL		:REAL := 0.2;
	HALTED_VEL_TOL		:REAL := 1.0;
END_VAR

(*
	FB_CTC_PlcOpen V3.0
	Cyltronic AG, September 2024

	Function Block that handles an CTC/L/R IO-Link Cylinder, based on Standard Motion
	Block (PLCOpen)

	V3.0: Added brake functionality

	Cyltronic Firmware compatibility:
	< V2.06.02: This version only has the option "Home Mode Direct", so it's not really 
				usable with this Function Block, as the user can only teach or home direct
	= V2.06.02: This FW version has no "Enable" functionality, so it's not compatible
				with a break mode. DO NOT USE WITH BREAK MODE
	> V2.06.02: Compatible with break mode

	NOTE:
	stConfiguration must match Cyltronic drive acyclic configuration parameters, 
	otherwise this function block will not work as intended
*)

// =================================================================================
// === PROCESS DATA INPUTS =========================================================
// =================================================================================
// Status = Byte 0
stProcessDataIn.State := BYTE_TO_USINT(ProcessDataInRaw[0]);
// StatusBits = Byte 1
stProcessDataIn.stStatusBits.TrackingErrorToleranceExceeded	:= ProcessDataInRaw[1].7;
stProcessDataIn.stStatusBits.WarningActive 					:= ProcessDataInRaw[1].6;
stProcessDataIn.stStatusBits.MotionCommandCompleted 		:= ProcessDataInRaw[1].5;
stProcessDataIn.stStatusBits.MotionModeActive 				:= ProcessDataInRaw[1].4;
stProcessDataIn.stStatusBits.LimitSwitchIn 					:= ProcessDataInRaw[1].3;
stProcessDataIn.stStatusBits.LimitSwitchOut 				:= ProcessDataInRaw[1].2;
stProcessDataIn.stStatusBits.Homed 							:= ProcessDataInRaw[1].1;
stProcessDataIn.stStatusBits.Ready 							:= ProcessDataInRaw[1].0;
// Actual Position = Bytes 2-5
unionContainer.aBytes[0] := ProcessDataInRaw[5];
unionContainer.aBytes[1] := ProcessDataInRaw[4];
unionContainer.aBytes[2] := ProcessDataInRaw[3];
unionContainer.aBytes[3] := ProcessDataInRaw[2];
stProcessDataIn.ActualPosition := unionContainer.rReal;
// Actual Speed = Bytes 6-9
unionContainer.aBytes[0] := ProcessDataInRaw[9];
unionContainer.aBytes[1] := ProcessDataInRaw[8];
unionContainer.aBytes[2] := ProcessDataInRaw[7];
unionContainer.aBytes[3] := ProcessDataInRaw[6];
stProcessDataIn.ActualSpeed := unionContainer.rReal;
// Actual Force = Bytes 10-13
unionContainer.aBytes[0] := ProcessDataInRaw[13];
unionContainer.aBytes[1] := ProcessDataInRaw[12];
unionContainer.aBytes[2] := ProcessDataInRaw[11];
unionContainer.aBytes[3] := ProcessDataInRaw[10];
stProcessDataIn.ActualForce := unionContainer.rReal;

// =================================================================================
// === Catch rising edges ==========================================================
// =================================================================================
// Some commands only valid on rising edges, so we catch these and set internal commands
R_TRIG_Array[0](CLK := Halt);
IF (R_TRIG_Array[0].Q) THEN
stInternalCommands.bHalt := TRUE;
ELSIF (NOT Halt) THEN
    stInternalCommands.bHalt := FALSE;
END_IF;

R_TRIG_Array[1](CLK := Home);
IF (R_TRIG_Array[1].Q) THEN
    stInternalCommands.bHome := TRUE;
ELSIF (NOT Home) THEN
    stInternalCommands.bHome := FALSE;
END_IF;

R_TRIG_Array[2](CLK := Teach);
IF (R_TRIG_Array[2].Q) THEN
    stInternalCommands.bTeach := TRUE;
ELSIF (NOT Teach) THEN
    stInternalCommands.bTeach := FALSE;
END_IF;

R_TRIG_Array[3](CLK := MoveAbsolute);
IF (R_TRIG_Array[3].Q) THEN
    stInternalCommands.bMoveAbsolute := TRUE;
ELSIF (NOT MoveAbsolute) THEN
    stInternalCommands.bMoveAbsolute := FALSE;
END_IF;

R_TRIG_Array[4](CLK := MoveContinuous);
IF (R_TRIG_Array[4].Q) THEN
    stInternalCommands.bMoveContinuous := TRUE;
ELSIF (NOT MoveContinuous) THEN
    stInternalCommands.bMoveContinuous := FALSE;
END_IF;

R_TRIG_Array[5](CLK := MoveIn);
IF (R_TRIG_Array[5].Q) THEN
    stInternalCommands.bMoveIn := TRUE;
ELSIF (NOT MoveIn) THEN
    stInternalCommands.bMoveIn := FALSE;
END_IF;

R_TRIG_Array[6](CLK := MoveOut);
IF (R_TRIG_Array[6].Q) THEN
	stInternalCommands.bMoveOut := TRUE;
ELSIF (NOT MoveOut) THEN
    stInternalCommands.bMoveOut := FALSE;
END_IF;

// =================================================================================
// === CTC State Machine ===========================================================
// =================================================================================
// Global guards which force state machine into defined states	
IF(Enable = FALSE)THEN
	stProcessDataOut.MotionMode := CTC_MOTION_MODE_OFF;
	eStep := FB_CTC_FUNCTIONBLOCK_DISABLED;
ELSIF(eStep > FB_CTC_CONNECTING AND stProcessDataIn.State = CTC_STATUS_BYTE_IDLE)THEN
	eStep := FB_CTC_FUNCTIONBLOCK_DISABLED;
END_IF
IF (Enable = FALSE) THEN
    stProcessDataOut.MotionMode := CTC_MOTION_MODE_OFF;
    eStep := FB_CTC_FUNCTIONBLOCK_DISABLED;
END_IF;

CASE eStep OF
        // ========================================================
        // === FB FUNCTIONBLOCK DISABLED ==========================
        // ========================================================
    FB_CTC_FUNCTIONBLOCK_DISABLED:
        
        stProcessDataOut.MotionMode := CTC_MOTION_MODE_OFF;
		ReleaseBrake := FALSE;
		
		Busy := FALSE;
		Done := FALSE;
		Error := FALSE;
        
        IF (Enable = TRUE) THEN
            eStep := FB_CTC_CONNECTING;
        END_IF;
        
        // ========================================================
        // === FB_CTC_CONNECTING ==================================
        // ========================================================
    FB_CTC_CONNECTING:
        
        IF (stProcessDataIn.State = CTC_STATUS_BYTE_READY) THEN
            eStep := FB_CTC_DISABLED;
        ELSIF (Reset = TRUE) THEN
            eStep := FB_CTC_RESET;
        ELSIF (stProcessDataIn.State = CTC_STATUS_BYTE_ERROR) THEN
            Busy := FALSE;
            Done := FALSE;
            Error := TRUE;
            stProcessDataOut.MotionMode := CTC_MOTION_MODE_HALT;
            eStep := FB_CTC_ERROR;
        END_IF;
        
        // ========================================================
        // === DISABLED ===========================================
        // ========================================================
    FB_CTC_DISABLED:
        
        stProcessDataOut.MotionMode := CTC_MOTION_MODE_OFF;
        
        Busy := FALSE;
        Done := FALSE;
        Error := FALSE;
        
		IF((Power = TRUE) AND (stProcessDataIn.State = CTC_STATUS_BYTE_READY))THEN
				
			// homed drive may be powered on...
			IF(stProcessDataIn.stStatusBits.Homed = TRUE)THEN
				
				// we power on by setting targetpos=actualpos, with a tolerance when we are near the configured end positions
				IF(stProcessDataIn.ActualPosition < stConfiguration.EndPositionIn 
					AND stProcessDataIn.ActualPosition >= (stConfiguration.EndPositionIn - FREE_POS_TOL))THEN
					stProcessDataOut.TargetPosition := stConfiguration.EndPositionIn;
				ELSIF(stProcessDataIn.ActualPosition > stConfiguration.EndPositionOut 
					AND stProcessDataIn.ActualPosition <= (stConfiguration.EndPositionOut + FREE_POS_TOL))THEN
					stProcessDataOut.TargetPosition := stConfiguration.EndPositionOut;
				ELSE
					stProcessDataOut.TargetPosition := stProcessDataIn.ActualPosition;
				END_IF
				
				stProcessDataOut.MotionMode := CTC_MOTION_MODE_FREEPOS;
				
				TON_Brake.IN := FALSE;
				eStep := FB_CTC_ENABLING;
				
			ELSE
				// ... unhomed drive stays powered off and brake stays active
				eStep := FB_CTC_READY;
			END_IF
			ELSE
			stProcessDataOut.MotionMode := CTC_MOTION_MODE_OFF;
		END_IF
       
        // === Catch error
        IF (stProcessDataIn.State = CTC_STATUS_BYTE_ERROR) THEN
            Busy := FALSE;
            Done := FALSE;
            Error := TRUE;
            stProcessDataOut.MotionMode := CTC_MOTION_MODE_HALT;
            eStep := FB_CTC_ERROR;
        END_IF;
        
		
		// ========================================================
		// === ENABLING ===========================================
		// ========================================================
	FB_CTC_ENABLING:
		
		// delay releasing brake according brake mode. Wait for drive status active
		IF(BrakeMode = CTC_BRAKE_MODE_WHEN_DISABLED)THEN
			TON_Brake.PT := UINT_TO_TIME(BrakeDelay);
			TON_Brake.IN := TRUE;
			IF(TON_Brake.Q AND (stProcessDataIn.State = CTC_STATUS_BYTE_ACTIVE))THEN
				TON_Brake.IN := FALSE;
				ReleaseBrake := TRUE;
				eStep := FB_CTC_READY;
			END_IF
		ELSIF(stProcessDataIn.State = CTC_STATUS_BYTE_ACTIVE)THEN
			TON_Brake.IN := FALSE;
			ReleaseBrake := FALSE;
			eStep := FB_CTC_READY;	
		END_IF
		
		// === Catch power off or halt
		IF(Power = FALSE)THEN
			stProcessDataOut.MotionMode := CTC_MOTION_MODE_OFF;
			eStep := FB_CTC_DISABLED;
		END_IF
		
		// === Catch error
		IF(stProcessDataIn.State = CTC_STATUS_BYTE_ERROR)THEN
			Busy 	:= FALSE;
			Done	:= FALSE;
			Error 	:= TRUE;
			stProcessDataOut.MotionMode := CTC_MOTION_MODE_HALT;
			eStep := FB_CTC_ERROR;
		END_IF
		
		// ========================================================
		// === DISABLING ==========================================
		// ========================================================
	FB_CTC_DISABLING:
		
		IF((BrakeMode = CTC_BRAKE_MODE_WHEN_DISABLED) AND Homed)THEN
			
			CASE iIntermediateStep OF
				0: // if brake option is active, try to at least halt drive until brake enables...
					stProcessDataOut.MotionMode := CTC_MOTION_MODE_HALT;
					TON_Brake.PT := UINT_TO_TIME(BrakeDelay);
					TON_Brake.IN := TRUE;
					IF(TON_Brake.Q)THEN
						TON_Brake.IN := FALSE;
						ReleaseBrake := FALSE;
						iIntermediateStep := 1;
					END_IF
				1: // ...and after another delay, drive disables
					TON_Brake.PT := UINT_TO_TIME(BrakeDelay);
					TON_Brake.IN := TRUE;
					IF(TON_Brake.Q)THEN
						TON_Brake.IN := FALSE;
						iIntermediateStep := 2;
						stProcessDataOut.MotionMode := CTC_MOTION_MODE_OFF;
					END_IF
					
				2: // transition only if drive has been deactivated successfully
					IF(stProcessDataIn.State = CTC_STATUS_BYTE_READY)THEN
						TON_Brake.IN := FALSE;
						iIntermediateStep := 0;
						eStep := FB_CTC_DISABLED;
					END_IF
					
				ELSE
					iIntermediateStep := 0;
			END_CASE;
			
		ELSE // if no brake, or the drive is not homed (meaning not powered on), 
			// then drive is disabled immediately. Transition only if drive has been deactivated successfully
			stProcessDataOut.MotionMode := CTC_MOTION_MODE_OFF;
			IF(stProcessDataIn.State = CTC_STATUS_BYTE_READY)THEN
				TON_Brake.IN := FALSE;
				iIntermediateStep := 0;
				eStep := FB_CTC_DISABLED;
			END_IF
		END_IF
			
        // ====================================================
        // === READY ==========================================
        // ====================================================
    FB_CTC_READY:
        
        TON_MMComplete.IN := 0;
        iIntermediateStep := 0;
        
        Busy := FALSE;
        Done := FALSE;
        
        IF (stInternalCommands.bHome = TRUE) THEN
            stInternalCommands.bHome := FALSE;
            bSetpointError := FALSE;
            Busy := TRUE;
            Done := FALSE;
            stProcessDataOut.MotionMode := CTC_MOTION_MODE_HALT;
            eStep := FB_CTC_HOME;
        ELSIF (stInternalCommands.bTeach = TRUE) THEN
            stInternalCommands.bTeach := FALSE;
            Busy := TRUE;
            Done := FALSE;
            bSetpointError := FALSE;
            stProcessDataOut.MotionMode := CTC_MOTION_MODE_HALT;
            eStep := FB_CTC_TEACH;
        ELSIF (stInternalCommands.bMoveIn = TRUE) THEN
            stInternalCommands.bMoveIn := FALSE;
            //IF (Homed) THEN
                Busy := TRUE;
                Done := FALSE;
                bSetpointError := FALSE;
                eStep := FB_CTC_MOVE_IN;
            //END_IF;
        ELSIF (stInternalCommands.bMoveOut = TRUE) THEN
            stInternalCommands.bMoveOut := FALSE;
            //IF (Homed) THEN
                Busy := TRUE;
                Done := FALSE;
                bSetpointError := FALSE;
                eStep := FB_CTC_MOVE_OUT;
            //END_IF;
        ELSIF (stInternalCommands.bMoveAbsolute = TRUE) THEN
            stInternalCommands.bMoveAbsolute := FALSE;
            IF (Homed) THEN
                Busy := TRUE;
                Done := FALSE;
                bSetpointError := FALSE;
                eStep := FB_CTC_MOVE_ABSOLUTE;
            END_IF;
        ELSIF (stInternalCommands.bMoveContinuous = TRUE) THEN
            IF (Homed) THEN
                Busy := TRUE;
                Done := FALSE;
                bSetpointError := FALSE;
                eStep := FB_CTC_MOVE_CONTINUOUS;
            END_IF;
        END_IF;
        
        // === Catch power off or halt
        IF (Power = FALSE) THEN
			TON_Brake.IN := FALSE;
			iIntermediateStep := 0;
			eStep := FB_CTC_DISABLING;
        ELSIF (stInternalCommands.bHalt = TRUE) THEN
            stInternalCommands.bHalt := FALSE;
            stProcessDataOut.MotionMode := CTC_MOTION_MODE_HALT;
            eStep := FB_CTC_HALTING;
        END_IF;
        
        // === Catch error
        IF (stProcessDataIn.State = CTC_STATUS_BYTE_ERROR) THEN
            Busy := FALSE;
            Done := FALSE;
            Error := TRUE;
            stProcessDataOut.MotionMode := CTC_MOTION_MODE_HALT;
            eStep := FB_CTC_ERROR;
        END_IF;
        
        // ====================================================
        // === HOME ===========================================
        // ====================================================
    FB_CTC_HOME:
			
		CASE iIntermediateStep OF
							
			0: 	// we can start homing if brake mode is off, or if brake is already released...
				IF(BrakeMode = CTC_BRAKE_MODE_OFF OR (ReleaseBrake = TRUE))THEN
					iIntermediateStep := 21;
				ELSE
					// ...else we must enable drive and release brake first
					stProcessDataOut.MotionMode := CTC_MOTION_MODE_HALT;
					TON_Brake.IN := FALSE;
					iIntermediateStep := 11;
				END_IF
				
			11: // delay --> release brake (check for active drive) --> 12
				TON_Brake.PT := UINT_TO_TIME(BrakeDelay);
				TON_Brake.IN := TRUE;
				IF(TON_Brake.Q AND (stProcessDataIn.State = CTC_STATUS_BYTE_ACTIVE))THEN
					TON_Brake.IN := FALSE;
					ReleaseBrake := TRUE;
					iIntermediateStep := 12;
				END_IF
				
			12: // delay --> start homing --> 21
				TON_Brake.PT := UINT_TO_TIME(BrakeDelay);
				TON_Brake.IN := TRUE;
				IF(TON_Brake.Q)THEN
					TON_Brake.IN := FALSE;
					iIntermediateStep := 21;
				END_IF
				
			21:	// home mode dependant on actual configuration					
				IF (stConfiguration.HomeMode = CTC_HOME_MODE_ENDSTOPIN) THEN
					iIntermediateStep := 22;
				ELSIF (stConfiguration.HomeMode = CTC_HOME_MODE_ENDSTOPOUT) THEN
					iIntermediateStep := 23;
				ELSE
					stProcessDataOut.TargetPosition := stParameters.TargetPosition;
					iIntermediateStep := 24;
				END_IF
				stProcessDataOut.MotionMode := CTC_MOTION_MODE_HOME;
				
			22:	// Home in
				IF((stProcessDataIn.stStatusBits.Homed = TRUE) AND 
					(stProcessDataIn.stStatusBits.LimitSwitchIn = TRUE OR stProcessDataIn.stStatusBits.LimitSwitchOut = TRUE))THEN
					Busy := FALSE;
					Done := TRUE;
					stProcessDataOut.MotionMode := CTC_MOTION_MODE_HALT;
					iIntermediateStep := 0;
					eStep := FB_CTC_READY;
				END_IF
				
			23: // Home out
				IF((stProcessDataIn.stStatusBits.Homed = TRUE) AND 
					(stProcessDataIn.stStatusBits.LimitSwitchIn = TRUE OR stProcessDataIn.stStatusBits.LimitSwitchOut = TRUE))THEN
					Busy := FALSE;
					Done := TRUE;
					stProcessDataOut.MotionMode := CTC_MOTION_MODE_HALT;
					iIntermediateStep := 0;
					eStep := FB_CTC_READY;
				END_IF
			
			24: // Home direct
				Busy := FALSE;
				Done := TRUE;
				stProcessDataOut.MotionMode := CTC_MOTION_MODE_HOME;
				iIntermediateStep := 0;
				eStep := FB_CTC_READY;
				
			ELSE
				iIntermediateStep := 0;
			
		END_CASE;
		
		// ---
		bHomeTeachFailed := stProcessDataIn.State = CTC_STATUS_BYTE_TEACH 
		AND stProcessDataIn.stStatusBits.WarningActive 
		AND NOT stProcessDataIn.stStatusBits.TrackingErrorToleranceExceeded;
		// ---
		
		// === Catch power off or halt
		IF(Power = FALSE)THEN	
			TON_Brake.IN := FALSE;
			iIntermediateStep := 0;
			eStep := FB_CTC_DISABLING;
		ELSIF(stInternalCommands.bHalt = TRUE OR bHomeTeachFailed)THEN
			stInternalCommands.bHalt := FALSE;
			stProcessDataOut.MotionMode := CTC_MOTION_MODE_OFF;
			IF(BrakeMode = CTC_BRAKE_MODE_WHEN_DISABLED)THEN
				ReleaseBrake := FALSE;
			END_IF
			eStep := FB_CTC_DISABLED;
		END_IF
			// === Catch error
		IF(stProcessDataIn.State = CTC_STATUS_BYTE_ERROR)THEN
			Busy 	:= FALSE;
			Done	:= FALSE;
			Error 	:= TRUE;
			stProcessDataOut.MotionMode := CTC_MOTION_MODE_HALT;
			eStep := FB_CTC_ERROR;
		END_IF
	        
       // ====================================================
       // === TEACH ==========================================
       // ====================================================
	FB_CTC_TEACH:
				
		// TEACH IS NOT COMPATIBLE WITH BRAKE & OLDER FW (<= V2.06.02!)
		
		CASE iIntermediateStep OF
				
			0: 	// if no brake, we can start teach via Mode 0 (compatible with older FW)
				// if brake, but released, then teach via Mode 1 (not compatible with older FW)
				// if brake, but not released --> enable drive, release brake, teach via Mode 1 (not compatible with older FW)
				IF(BrakeMode = CTC_BRAKE_MODE_OFF)THEN
					stProcessDataOut.MotionMode := CTC_MOTION_MODE_OFF;
					iIntermediateStep := 21;
				ELSIF(ReleaseBrake = TRUE)THEN
					stProcessDataOut.MotionMode := CTC_MOTION_MODE_HALT; // this enables drive
					iIntermediateStep := 21;
				ELSE
					stProcessDataOut.MotionMode := CTC_MOTION_MODE_HALT; // this enables drive
					TON_Brake.IN := FALSE;
					iIntermediateStep := 11;
				END_IF
				
			11: // delay --> release brake (if drive active) --> 12
				TON_Brake.PT := UINT_TO_TIME(BrakeDelay);
				TON_Brake.IN := TRUE;
				IF(TON_Brake.Q AND (stProcessDataIn.State = CTC_STATUS_BYTE_ACTIVE))THEN // older drives will get stuck here, so the break will not release
					TON_Brake.IN := FALSE;
					ReleaseBrake := TRUE;
					iIntermediateStep := 12;
				END_IF
				
			12: // delay --> start teaching --> 21
				TON_Brake.PT := UINT_TO_TIME(BrakeDelay);
				TON_Brake.IN := TRUE;
				IF(TON_Brake.Q)THEN
					TON_Brake.IN := FALSE;
					iIntermediateStep := 21;
				END_IF
				
			21: // teach only allowed out of "off" and "ready, i.e. ready state
				IF((stProcessDataIn.State = CTC_STATUS_BYTE_READY) OR (stProcessDataIn.State = CTC_STATUS_BYTE_ACTIVE))THEN
					stProcessDataOut.MotionMode := CTC_MOTION_MODE_TEACH;
					iIntermediateStep := 22;
				END_IF				
			22:				
				IF(stProcessDataIn.State = CTC_STATUS_BYTE_TEACH)THEN
					iIntermediateStep := 23;
				END_IF
			23:
				IF(stProcessDataIn.State <> CTC_STATUS_BYTE_TEACH)THEN
					Busy := FALSE;
					Done := TRUE;
					stProcessDataOut.MotionMode := CTC_MOTION_MODE_HALT;
					eStep := FB_CTC_READY;
					iIntermediateStep := 0;
				END_IF
				
			ELSE
				iIntermediateStep := 0;
		END_CASE
		
		// ---
		bHomeTeachFailed := stProcessDataIn.State = CTC_STATUS_BYTE_TEACH 
		AND stProcessDataIn.stStatusBits.WarningActive 
		AND NOT stProcessDataIn.stStatusBits.TrackingErrorToleranceExceeded;
		// ---
		
		// === Catch power off or halt
		IF(Power = FALSE)THEN
			TON_Brake.IN := FALSE;
			iIntermediateStep := 0;
			eStep := FB_CTC_DISABLING;			
		ELSIF(stInternalCommands.bHalt = TRUE OR bHomeTeachFailed)THEN
			stInternalCommands.bHalt := FALSE;
			stProcessDataOut.MotionMode := CTC_MOTION_MODE_OFF;
			IF(BrakeMode = CTC_BRAKE_MODE_WHEN_DISABLED)THEN
				ReleaseBrake := FALSE;
			END_IF
			eStep := FB_CTC_DISABLED;
		END_IF
		// === Catch error
		IF(stProcessDataIn.State = CTC_STATUS_BYTE_ERROR)THEN
			Busy 	:= FALSE;
			Done	:= FALSE;
			Error 	:= TRUE;
			stProcessDataOut.MotionMode := CTC_MOTION_MODE_HALT;
			eStep := FB_CTC_ERROR;
		END_IF
		
		
		// ====================================================
		// === MOVEOUT ========================================
		// ====================================================
	FB_CTC_MOVE_OUT:
		
		TON_MMComplete.IN := stProcessDataIn.stStatusBits.MotionCommandCompleted;					
		stProcessDataOut.MotionMode := CTC_MOTION_MODE_MOVEOUT;
		
		IF((stProcessDataIn.stStatusBits.LimitSwitchOut = TRUE) AND (TON_MMComplete.Q = TRUE))THEN
			Busy := FALSE;
			Done := TRUE;
			stProcessDataOut.MotionMode := CTC_MOTION_MODE_HALT;
			eStep := FB_CTC_READY;
		END_IF
			// === Catch power off or halt or state transition
		IF(Power = FALSE)THEN
			TON_Brake.IN := FALSE;
			iIntermediateStep := 0;
			eStep := FB_CTC_DISABLING;
		ELSIF(stInternalCommands.bHalt = TRUE)THEN
			stInternalCommands.bHalt := FALSE;
			stProcessDataOut.MotionMode := CTC_MOTION_MODE_HALT;
			eStep := FB_CTC_HALTING;
		ELSIF(stInternalCommands.bMoveIn OR stInternalCommands.bMoveAbsolute 
			OR stInternalCommands.bMoveContinuous)THEN
			eStep := FB_CTC_READY;
		END_IF
		
			// === Catch error
		IF(stProcessDataIn.State = CTC_STATUS_BYTE_ERROR)THEN
			Busy 	:= FALSE;
			Done	:= FALSE;
			Error 	:= TRUE;
			stProcessDataOut.MotionMode := CTC_MOTION_MODE_HALT;
			eStep := FB_CTC_ERROR;
		END_IF
		      
      	// ====================================================
      	// === MOVEIN =========================================
		// ====================================================
	FB_CTC_MOVE_IN:
        
        TON_MMComplete.IN := stProcessDataIn.stStatusBits.MotionCommandCompleted;
        stProcessDataOut.MotionMode := CTC_MOTION_MODE_MOVEIN;
        
        IF ((stProcessDataIn.stStatusBits.LimitSwitchIn = TRUE) AND (TON_MMComplete.Q = TRUE)) THEN
            Busy := FALSE;
            Done := TRUE;
            stProcessDataOut.MotionMode := CTC_MOTION_MODE_HALT;
            eStep := FB_CTC_READY;
        END_IF;
        
